(* CODESYS project sensata_vision.library
   Company: Sensata Technologies
   Version: 0.0.2
   DocFormat: reStructuredText
   Placeholder: Sensata_Vision
   Title: Sensata_Vision

Project tree, tasks and I/O mapping:
  libraries: Sensata_Common, * (Sensata Technologies); Sensata_IO, * (Sensata Technologies); Tc2_Standard, * (Beckhoff Automation GmbH); Tc2_System, * (Beckhoff Automation GmbH); Tc2_Utilities, * (Beckhoff Automation GmbH); Tc3_Module, * (Beckhoff Automation GmbH)
  Abstract/
    function block FB_BarcodeReader [ST]
    function block FB_Camera [ST]: M_SaveImage, P_bSaveImageBusy, M_ClearResults, M_ReadResult, P_bReadBusy, P_bResultsAvailable, M_Trigger, P_bTriggerBusy
  Concrete/
    Cognex/
      D900/
        data type E_CognexD900_Error
        function block FB_CognexD900 [ST]: P_strDescription, P_strMake, P_strModel, P_strVersion, M_Disable, M_Enable, M_GetEnableStatus, P_bEnableBusy, P_bEnabled, M_SaveImage, P_bSaveImageBusy, M_GetCurrentProgram, M_GetProgramState, M_LoadProgram, M_PauseProgram, M_StartProgram, M_StopProgram, P_bProgramControlBusy, P_enumProgramState, P_strCurrentProgram, M_ClearResults, M_ReadResult, P_bReadBusy, P_bResultsAvailable, M_Reset, P_bResetBusy, M_Trigger, P_bTriggerBusy
        data type ST_CognexD900_IO_Inputs
        data type ST_CognexD900_IO_Outputs
    Keyence/
      IX Series/
        function block FB_KeyenceIX_DLEC1A [ST]: M_Reset, P_bResetBusy, M_Trigger, P_bTriggerBusy, A_CommandRecovery, A_ControlsMapping, A_ValueMapping
        data type ST_KeyenceIXValue
      SR Series/
        Old/
          function block FB_KeyenceBarcodeReader [ST]: M_Disable, M_Enable, M_GetCurrentProgram, M_GetEnableStatus, M_GetProgramState, M_LoadProgram, M_PauseProgram, M_ReadResults, M_Reset, M_StartProgram, M_StopProgram, M_Trigger, P_bEnableBusy, P_bEnabled, P_bProgramControlBusy, P_bReadBusy, P_bResetBusy, P_bResultsAvailable, P_bTriggerBusy, P_enumProgramState, P_strCurrentProgram, P_strDescription, P_strMake, P_strModel, P_strVersion
          data type KeyenceSR700_Inputs
          data type KeyenceSR700_Outputs
        function block FB_KeyenceNL20_EIP [ST]: A_SR, M_ClearResults, M_ReadResult, M_Reset, M_Trigger, P_bReadBusy, P_bResetBusy, P_bResultsAvailable, P_bTriggerBusy
        function block FB_KeyenceSR [ST]: M_ClearResults, M_ReadResult, P_bReadBusy, P_bResultsAvailable, M_Reset, P_bResetBusy, M_Trigger, P_bTriggerBusy, A_ClearOutputs, A_CommandRecovery
        function block FB_KeyenceSR750_EIP [ST]: A_SR, M_ClearResults, M_ReadResult, M_Reset, M_Trigger, P_bReadBusy, P_bResetBusy, P_bResultsAvailable, P_bTriggerBusy
        function block FB_KeyenceSRX1H3H_EIP [ST]: A_SR, M_ClearResults, M_ReadResult, M_Reset, M_Trigger, P_bReadBusy, P_bResetBusy, P_bResultsAvailable, P_bTriggerBusy
  Interfaces/
    interface I_ImageSaving: M_SaveImage, P_bSaveImageBusy
    interface I_Readable: M_ClearResults, M_ReadResult, P_bReadBusy, P_bResultsAvailable
    interface I_Triggerable: M_Trigger, P_bTriggerBusy
  Project Information/
    function F_GetCompany [ST]
    function F_GetTitle [ST]
    function F_GetVersion [ST]
  Version/
    global variables Global_Version
*)

// Concrete/Cognex/D900/E_CognexD900_Error
{attribute 'qualified_only'}
{attribute 'strict'}
TYPE E_CognexD900_Error :
(
	NoError := 0,
	
	LoadProgramFail := 100,
	LoadRecipeFail := 101,
	
	TriggerTimeout := 200,
	
	ImageNameOrLocationTooLong := 300
) UDINT;
END_TYPE

// Concrete/Cognex/D900/ST_CognexD900_IO_Inputs
TYPE ST_CognexD900_IO_Inputs :
STRUCT
	bOnline : BOOL; (* Standard input from camera. TRUE when the camera is online. *)
	bReady : BOOL; (* Standard input from camera. TRUE when the camera is ready. *)
	bPaused : BOOL; (* Standard input from camera. TRUE when the camera is paused. *)
	bHasError : BOOL; (* Standard input from camera. TRUE when the camera has an error. *)
	intErrorCode : INT; (* Standard input from camera. Current error code. *)
	
	bTriggerReady : BOOL; (* Standard input from camera. TRUE when the trigger is ready. *)
	bTriggerAck : BOOL; (* Standard input from camera. Goes TRUE to acknowledge a trigger. *)
	bAcquisitionError : BOOL; (* Standard input from camera. Goes TRUE if acquisition failed. *)
	bExposureComplete : BOOL; (* Standard input from camera. Goes TRUE if exposure finished. *)
	
	bResultsValid : BOOL; (* Standard input from camera. Goes TRUE once inspection results are available. *)
	
	bCommandFailed : BOOL; (* Standard input from camera. TRUE if a command has failed. *)
	bCommandCompleted : BOOL; (* Standard input from camera. TRUE if a command has completed. *)
	
	bSetUserDataAck :  BOOL; (* Standard input from camera. Goes TRUE to acknowledge setting of user data buffer. *)

	bReadUserDataAck : BOOL; (* Should be assigned to an external trigger if image saving is used. *)
	bSaveImageAck : BOOL; (* Should be assigned to an external trigger if image saving is used. *)
END_STRUCT
END_TYPE

// Concrete/Cognex/D900/ST_CognexD900_IO_Outputs
TYPE ST_CognexD900_IO_Outputs :
STRUCT
	bTriggerEnable : BOOL; (* Standard output to camera. Set TRUE to enable trigger, FALSE to disable. *)
	bTrigger : BOOL; (* Standard output to camera. Rising edge to trigger camera. *)
	
	bResultAck : BOOL; (* Standard output to camera. Rising edge to acknowledge inspection result. *)
	
	bSetPaused : BOOL; (* Standard output to camera. Set TRUE to pause, FALSE to unpause. *)
	
	bClearError : BOOL; (* Standard output to camera. Rising edge to clear error. *)
	
	uintCommand : UINT; (* Standard output to camera. Set to a valid command ID before executing command. *)
	bExecuteCommand : BOOL; (* Standard output to camera. Set high to execute command. *)
	
	bSetUserData: BOOL; (* Standard output to camera. Set high to set user data buffer. *)
	
	bReadUserData : BOOL; (* Should be assigned to an external trigger if image saving is used. *)
	bSaveImage : BOOL; (* Should be set to an external trigger if image saving is enabled. *)
END_STRUCT
END_TYPE

// Concrete/Keyence/IX Series/ST_KeyenceIXValue
TYPE ST_KeyenceIXValue :
STRUCT
	bInvalid: BOOL;
	bUnderRange: BOOL;
	bOverRange: BOOL;
	dintValue: DINT;
END_STRUCT
END_TYPE

// Concrete/Keyence/SR Series/Old/KeyenceSR700_Inputs
TYPE KeyenceSR700_Inputs :
STRUCT
	Error								:BOOL;
	ResultDataAvailable					:BOOL;
	ResultDataStrobe					:BOOL;

	NoName0_arrBIT						:ARRAY[0..2] OF BOOL;
	NoName1_arrBIT						:ARRAY[0..2] OF BOOL;
	NoName2_arrBIT						:ARRAY[0..2] OF BOOL;
	NoName3_arrBIT						:ARRAY[0..2] OF BOOL;
	NoName4_arrBIT						:ARRAY[0..1] OF BOOL;
	NoName5_arrBIT						:BOOL;
	NoName6_arrBIT						:ARRAY[0..18] OF BOOL;

	NoName7_arrBYTE						:ARRAY[0..1] OF BYTE;
	NoName8_arrBYTE						:ARRAY[0..5] OF BYTE;
	NoName9_arrBYTE						:ARRAY[0..1] OF BYTE;
	NoName10_arrBYTE					:ARRAY[0..1] OF BYTE;


	BufferOverflowError					:BOOL;
	GeneralError						:BOOL;
	Busy								:BOOL;
	TRGBusy								:BOOL;
	LOCKBusy							:BOOL;
	ModeBusy							:BOOL;
	ErrorBusy							:BOOL;

	ReadComplete						:BOOL;
	PresetComplete						:BOOL;
	RegisterPresetDataComplete			:BOOL;
	TuneComplete						:BOOL;
	EXTRequestComplete					:BOOL;

	ReadFailure							:BOOL;
	PresetFailure						:BOOL;
	RegisterPresetDataFailure			:BOOL;
	TuneFailure							:BOOL;
	EXTRequestFailure					:BOOL;

	IN1Status							:BOOL;	
	IN2Status							:BOOL;	
	
	OUT1Status							:BOOL;	
	OUT2Status							:BOOL;	
	OUT3Status							:BOOL;	
		
	Unstable							:BOOL;
	MatchingLevel_Unstable				:BOOL;
	ISO_IEC15415_Unstable				:BOOL;
	AIM_DPM_Unstable					:BOOL;
	SAE_AS9132_Unstable					:BOOL;
	
	MatchingLevel						:UINT;
	ISO_IEC15415_Grade					:UINT;
	AIM_DPM_Grade						:UINT;

	ReadResultCode						:UINT;
	PresetResultCode					:UINT;
	RegisterPresetDataResultCode		:UINT;
	TuneResultCode						:UINT;
	EXTResquestResultCode				:UINT;
	GeneralErrorCode					:UINT;
	
	ResultData_ReadyCount				:UINT;
	ResultData_UpdateCount				:UINT;
	ResultData_Size						:UINT;
	ResultData							:ARRAY[0..128] OF BYTE;
	

END_STRUCT
END_TYPE

// Concrete/Keyence/SR Series/Old/KeyenceSR700_Outputs
TYPE KeyenceSR700_Outputs :
STRUCT

	ResultDataLatch						:BOOL;
	ClearError							:BOOL;

	ReadRequest							:BOOL;
	PresetRequest						:BOOL;
	RegisterPresetDataRequest			:BOOL;
	TuneRequest							:BOOL;

	ClearReadComplete					:BOOL;
	ClearPresetComplete					:BOOL;
	ClearRegisterPresetData				:BOOL;
	ClearTuneComplete					:BOOL;
	ClearEXTRequestComplete				:BOOL;

	BankNumber							:UINT;
	UserDataSize						:UINT;

	UserData							:ARRAY[0..64] OF BYTE;
	
	Noname0_BIT							:BOOL;
	Noname1_arrBIT						:ARRAY[0..4] OF BOOL;
	Noname2_arrBIT						:ARRAY[0..3] OF BOOL;
	Noname3_arrBIT						:ARRAY[0..2] OF BOOL;
	Noname4_BYTE						:BYTE;
	Noname5_arrBYTE						:ARRAY[0..3] OF BOOL;

END_STRUCT
END_TYPE

// Version/Global_Version
{attribute 'TcGenerated'}
{attribute 'no-analysis'}
{attribute 'linkalways'}
// This function has been automatically generated from the project information.
VAR_GLOBAL CONSTANT
	{attribute 'const_non_replaced'}
	stLibVersion_Sensata_Vision : ST_LibVersion := (iMajor := 0, iMinor := 0, iBuild := 2, iRevision := 0, nFlags := 0, sVersion := '0.0.2');
END_VAR

// Abstract/FB_BarcodeReader
FUNCTION_BLOCK ABSTRACT FB_BarcodeReader EXTENDS FB_Camera
VAR_INPUT
END_VAR
VAR_OUTPUT
END_VAR
VAR
END_VAR

END_FUNCTION_BLOCK

// Abstract/FB_Camera
(*
===============================================================================
Camera
===============================================================================
:Contact: Kevin Sanita <ksanita@sensata.com>
:Last Edited: December 2021

:Description: Represents a camera device.

:Notes:
* Standard use is to 
	1) Connect with I_Connectable
	2) Enable with I_Enableable
	3) Load program with I_Programmable
	4) Start program with I_Controllable
	5) While program is running, trigger with I_Triggerable
	6) Read inspect result with I_SimpleInspection

:Change Log:
- **December 20, 2021** Initial version
*)
FUNCTION_BLOCK ABSTRACT FB_Camera EXTENDS FB_Device
	IMPLEMENTS
		I_Triggerable, (* Most cameras will require triggering. *)
		I_Readable, (* Most cameras will require reading result data. *)
		I_ImageSaving (* Implements image saving functionality. *)
VAR_INPUT
END_VAR
VAR_OUTPUT
END_VAR
VAR
END_VAR

(* Saves an image with a specified name and save location. *)
METHOD M_SaveImage : BOOL
VAR_INPUT
	(* What to name the image file. *)
	strFilename	: Tc2_System.T_MaxString;
	(* Where to save the file, if applicable. *)
	strLocation	: Tc2_System.T_MaxString := '';
END_VAR
M_SaveImage := TRUE;
THIS^.M_LogWarning('M_SaveImage is not implemented!');
END_METHOD

PROPERTY P_bSaveImageBusy : BOOL
GET
P_bSaveImageBusy := FALSE;
END_GET
END_PROPERTY

(* Clears all results currently available on the camera. *)
METHOD M_ClearResults : BOOL
M_ClearResults := TRUE;
THIS^.M_LogWarning('Clear results not implemented!');
END_METHOD

(* Reads one result from the camera. *)
METHOD M_ReadResult : BOOL
M_ReadResult := TRUE;
THIS^.M_LogWarning('Read result not implemented!');
END_METHOD

(* True while this interface is busy. *)
PROPERTY P_bReadBusy : BOOL
GET
P_bReadBusy := FALSE;
END_GET
END_PROPERTY

(* True if there are results available. *)
PROPERTY P_bResultsAvailable : BOOL
GET
P_bResultsAvailable := FALSE;
END_GET
END_PROPERTY

(* Triggers the camera. *)
METHOD M_Trigger : BOOL
M_Trigger := TRUE;
THIS^.M_LogWarning('M_Trigger not implemented!');
END_METHOD

(* True while the camera is busy processing an image. *)
PROPERTY P_bTriggerBusy : BOOL
GET
P_bTriggerBusy := FALSE;
END_GET
END_PROPERTY

END_FUNCTION_BLOCK

// Interfaces/I_Triggerable
(*
===============================================================================
Triggerable
===============================================================================

:Description: Interface for modules that need to be triggered.

:Notes:
* Use ``M_Trigger`` to trigger the module.
* ``P_bTriggerBusy`` stays high while module is triggering. 
*)
INTERFACE I_Triggerable

(*
Triggers the function block.
*)
METHOD M_Trigger : BOOL
VAR_INPUT
END_VAR
END_METHOD

(*
Stays high while the function block is performing the tasks that were triggered.
*)
PROPERTY P_bTriggerBusy : BOOL
GET
END_GET
END_PROPERTY

END_INTERFACE

// Interfaces/I_Readable
(*
===============================================================================
Readable
===============================================================================

:Description: Interface for reading results data from inspection cameras.

:Notes:
* Use ``M_ReadResult`` to read result data from the camera.
* Use ``M_ClearResults`` to clear all results data.
* ``P_bReadBusy`` stays high while camera is being read. 
* ``P_bResultsAvailable`` is true if there is data available to read.
*)
INTERFACE I_Readable

(* Clears all results currently available on the camera. *)
METHOD M_ClearResults : BOOL
VAR_INPUT
END_VAR
END_METHOD

(* Reads one result from the camera. *)
METHOD M_ReadResult : BOOL
VAR_INPUT
END_VAR
END_METHOD

(* True while this interface is busy. *)
PROPERTY P_bReadBusy : BOOL
GET
END_GET
END_PROPERTY

(* True if there are results available. *)
PROPERTY P_bResultsAvailable : BOOL
GET
END_GET
END_PROPERTY

END_INTERFACE

// Interfaces/I_ImageSaving
INTERFACE I_ImageSaving

(* Saves an image with a specified name and save location. *)
METHOD M_SaveImage : BOOL
VAR_INPUT
	strFilename : T_MaxString; (* What to name the image file. *)
	strLocation : T_MaxString := ''; (* Where to save the file, if applicable. *)
END_VAR
END_METHOD

PROPERTY P_bSaveImageBusy : BOOL
GET
END_GET
END_PROPERTY

END_INTERFACE

// Concrete/Cognex/D900/FB_CognexD900
(*
===============================================================================
Function Block Name
===============================================================================
:Contact: Kevin Sanita <ksanita@sensata.com>
:Last Edited: January 2022

:Description: Cognex D900 implementation of FB_Camera

:Change Log:
- **January 4, 2021** Initial version
*)
FUNCTION_BLOCK FB_CognexD900 EXTENDS FB_Camera
	IMPLEMENTS 
		I_DeviceInfo, (* Required for all devices. *)
		I_Enableable, (* Cognex cameras have a trigger enable that must be set. *)
		I_Triggerable, (* The camera must be triggered to perform an inspection. *)
		I_Readable, (* Read results from the camera. *)
		I_Resettable, (* Need to be able to clear errors on the camera itself. *)
		I_Programmable, (* Must be able to load programs. *)
		I_ImageSaving (* Can use external triggers to save images. *)
VAR_INPUT
	stInputs : ST_CognexD900_IO_Inputs; (* Fieldbus inputs. *)
	arrUserData : REFERENCE TO ARRAY[0..487] OF BYTE; (* Standard output to camera. Contains user data for commands. *)
	
	(* Set to TRUE if image saving is enabled. Requires an event trigger to be
	set up in In-Sight Vision Suite. *)
	bImageSavingEnabled : BOOL; 
	uintImageFilenameOffset : UINT; (* User data location allocated to image filename. *)
	uintImageFilenameLength : UINT; (* User data length allocated to image filename. Set to zero to disable. *)
	uintImageLocationOffset : UINT; (* User data location allocated to image location. *)
	uintImageLocationLength : UINT; (* User data length allocated to image location. Set to zero to disable. *)
	
	// Program to load in format of job:recipe
	in_strProgram: T_MaxString;
END_VAR
VAR_OUTPUT
	stOutputs : ST_CognexD900_IO_Outputs; (* Fieldbus outputs. *)
END_VAR
VAR
	// Main
	fbErrorOccurred: R_TRIG; (* Rising edge trigger for errors. *)	

	// Control
	bControlBusy: BOOL; (* TRUE while pausing or unpausing camera program. *)
	
	// Trigger
	bTriggerBusy: BOOL; (* TRUE when the trigger is busy. *)
	
	// Read
	bReadBusy : BOOL; (* True while read is busy. *)
	
	// Reset
	bResetBusy: BOOL; (* TRUE when the camera is busy clearing error. *)
	
	// Load Program
	strRequestedProgram: STRING(255); (* The program request string containing job name or job and recipe separated by a colon. *)
	bProgramLoading: BOOL; (* TRUE while a job is loading. *)
	strRequestedJob: STRING(255); (* Requested job name. *)
	strRequestedRecipe: T_MaxString; (* Requested recipe name. *)
	intProgramLoadStep: INT; (* Current program loading step. *)
	intProgramRequestSplit: INT; (* Location of colon in program request string. *)
	strCurrentJob: T_MaxString; (* Currently loaded job *)
	strCurrentRecipe: T_MaxString; (* Currently loaded recipe. *)
	strCurrentProgram: T_MaxString; (* Currently loaded program. *)
	
	// Enable
	bEnableBusy: BOOL; (* TRUE while enable is busy. *)
	
	// Image saving
	bSaveImageBusy: BOOL; (* TRUE while image saving is busy. *)
	bUserDataSet: BOOL; (* TRUE if user data was set. *)
END_VAR

// Check camera for error.
fbErrorOccurred(CLK:=stInputs.bHasError);
IF fbErrorOccurred.Q THEN
	THIS^.M_SetError(INT_TO_UDINT(stInputs.intErrorCode), 'Camera error! Check camera documentation for error code details.');
END_IF

PROPERTY P_strDescription : Sensata_Common.T_MaxString
GET
P_strDescription := 'Cognex D900 Camera';
END_GET
END_PROPERTY

PROPERTY P_strMake : Sensata_Common.T_MaxString
GET
P_strMake := 'Cognex';
END_GET
END_PROPERTY

PROPERTY P_strModel : Sensata_Common.T_MaxString
GET
P_strModel := 'D900';
END_GET
END_PROPERTY

PROPERTY P_strVersion : Sensata_Common.T_MaxString
GET
END_GET
END_PROPERTY

(* Sets trigger enable low *)
METHOD M_Disable : BOOL
M_Disable := FALSE;
IF stOutputs.bTriggerEnable THEN
	bEnableBusy := TRUE;
	stOutputs.bTriggerEnable := FALSE;
	THIS^.M_LogMessage('Disabling trigger');
ELSIF NOT stInputs.bTriggerReady THEN
	IF bEnableBusy THEN
		bEnableBusy := FALSE;
		THIS^.M_LogMessage('Camera trigger disabled.');
	END_IF
	M_Disable := TRUE;
END_IF;
END_METHOD

(* Sets trigger enable high *)
METHOD M_Enable : BOOL
M_Enable := FALSE;
IF NOT stOutputs.bTriggerEnable THEN
	bEnableBusy := TRUE;
	stOutputs.bTriggerEnable := TRUE;
	THIS^.M_LogMessage('Enabling trigger');
ELSIF stInputs.bTriggerReady THEN
	IF bEnableBusy THEN
		bEnableBusy := FALSE;
		THIS^.M_LogMessage('Camera trigger enabled.');
	END_IF
	M_Enable := TRUE;
END_IF;
END_METHOD

(* Get the current enable status of the device. *)
METHOD M_GetEnableStatus : BOOL
VAR_OUTPUT
	bEnabled	: BOOL;
END_VAR
bEnabled := THIS^.P_bEnabled;
M_GetEnableStatus := TRUE;
END_METHOD

(* TRUE while the device is busy enabling or disabling. *)
PROPERTY P_bEnableBusy : BOOL
GET
P_bEnablebusy := bEnableBusy;
END_GET
END_PROPERTY

PROPERTY P_bEnabled : BOOL
GET
IF stInputs.bTriggerReady THEN
	P_bEnabled := TRUE;
ELSE
	P_bEnabled := FALSE;
END_IF
END_GET
END_PROPERTY

(* Saves an image with a specified name and save location. *)
METHOD M_SaveImage : BOOL
VAR_INPUT
	(* What to name the image file. *)
	strFilename	: Tc2_System.T_MaxString;
	(* Where to save the file, if applicable. *)
	strLocation	: Tc2_System.T_MaxString := '';
END_VAR

VAR
	bAbleToSave: BOOL;
	bFilenameValid: BOOL;
	bLocationValid: BOOL;
END_VAR
M_SaveImage := FALSE;

// Check that rest of camera isn't in a busy or error state
bAbleToSave := NOT THIS^.P_bError 
		AND NOT THIS^.P_bTriggerBusy
		AND NOT THIS^.P_bProgramControlBusy
		AND THIS^.P_enumProgramState = E_ProgramState.Running
		AND bImageSavingEnabled
		AND NOT bSaveImageBusy;

// If able to start saving, then try to start saving
IF bAbleToSave THEN
	
	// Check that the filename and location are not too long
	bFilenameValid := LEN(strFilename) < UINT_TO_INT(uintImageFilenameLength) OR uintImageFilenameLength = 0;
	bLocationValid := LEN(strLocation) < UINT_TO_INT(uintImageLocationLength) OR uintImageLocationLength = 0;
	
	IF bFilenameValid AND bLocationValid THEN
		// Send save image command
		bUserDataSet := FALSE;
		stOutputs.bSaveImage := FALSE;
		stOutputs.bSetUserData := FALSE;
		stOutputs.bReadUserData := FALSE;
		
		// Make sure the acknowledges are reset before starting trigger sequence
		IF NOT stInputs.bSaveImageAck AND NOT stInputs.bSetUserDataAck AND NOT stInputs.bReadUserDataAck THEN
			THIS^.M_LogMessage('Starting image save sequence.');
			bSaveImageBusy := TRUE;
		END_IF
	ELSE
		THIS^.M_SetError(
			E_CognexD900_Error.ImageNameOrLocationTooLong,
			'Filename or location for image saving is longer than allocated buffer space!');
	END_IF
	
// Wait for save image command to finish
ELSIF bSaveImageBusy THEN
	IF NOT bUserDataSet THEN
		IF NOT stOutputs.bSetUserData THEN
			// Save filename to user data buffer
			IF uintImageFilenameLength > 0 THEN
				MEMSET(ADR(arrUserData)+uintImageFilenameOffset, 0, uintImageFilenameLength);
				MEMCPY(ADR(arrUserData)+uintImageFilenameOffset, ADR(strFilename), INT_TO_UDINT(LEN(strFilename)));
			END_IF
			
			// Save location to user data sbuffer
			IF uintImageLocationLength > 0 THEN
				MEMSET(ADR(arrUserData)+uintImageLocationOffset, 0, uintImageLocationLength);
				MEMCPY(ADR(arrUserData)+uintImageLocationOffset, ADR(strLocation), INT_TO_UDINT(LEN(strLocation)));
			END_IF
		END_IF
		
		// Wait for user data to set.
		stOutputs.bSetUserData := TRUE;
		stOutputs.bReadUserData := TRUE;
		IF stInputs.bSetUserDataAck AND stInputs.bReadUserDataAck THEN
			THIS^.M_LogMessage('Set user data.');
			stOutputs.bReadUserData := FALSE;
			stOutputs.bSetUserData := FALSE;
			bUserDataSet := TRUE;
		END_IF
	ELSE
		// Wait for image to save
		stOutputs.bSaveImage := TRUE;
		IF stInputs.bSaveImageAck THEN
			THIS^.M_LogMessage('Image saved.');
			stOutputs.bSaveImage := FALSE;
			bSaveImageBusy := FALSE;
			M_SaveImage := TRUE;
		END_IF
	END_IF
END_IF
END_METHOD

PROPERTY P_bSaveImageBusy : BOOL
GET
P_bSaveImageBusy := bSaveImageBusy;
END_GET
END_PROPERTY

(* Gets the program currently loaded on the device. *)
METHOD M_GetCurrentProgram : BOOL
VAR_OUTPUT
	strCurrentProgram	: Sensata_Common.T_MaxString;
END_VAR
strCurrentProgram := THIS^.P_strCurrentProgram;
M_GetCurrentProgram := TRUE;
END_METHOD

(* Gets the current control state. *)
METHOD M_GetProgramState : BOOL
VAR_OUTPUT
	enumProgramState	: Sensata_Common.E_ProgramState;
END_VAR
enumProgramState := THIS^.P_enumProgramState;
M_GetProgramState := TRUE;
END_METHOD

 (*
Loads a new program on the module.
*)
METHOD M_LoadProgram : BOOL
M_LoadProgram := FALSE;

CASE intProgramLoadStep OF
	0: // Parse job and recipe
		bProgramLoading := TRUE;
		strRequestedProgram := in_strProgram;
		intProgramRequestSplit := FIND(strRequestedProgram, ':');
		IF intProgramRequestSplit > 0 THEN
			strRequestedJob := LEFT(strRequestedProgram, intProgramRequestSplit-1);
			strRequestedRecipe := RIGHT(strRequestedProgram, LEN(strRequestedProgram)-intProgramRequestSplit);
		ELSE
			strRequestedJob := strRequestedProgram;
			strRequestedRecipe := '';
		END_IF
		
		strCurrentProgram := '';
		
		intProgramLoadStep := intProgramLoadStep + 10;

	10: // Pause the camera
		IF THIS^.M_PauseProgram() THEN
			intProgramLoadStep := intProgramLoadStep + 10;
		END_IF
		
	20: // Send the load job by name command
		IF strCurrentJob <> strRequestedJob THEN
			// Set command to load program by name
			stOutputs.uintCommand := 16#4000; 

			// Copy program name to user data
			MEMSET(ADR(arrUserData), 0, SIZEOF(arrUserData));
			MEMCPY(ADR(arrUserData), ADR(strRequestedJob), INT_TO_UDINT(LEN(strRequestedJob)));
			
			// Set execute command bit
			stOutputs.bExecuteCommand := TRUE;
			
			THIS^.M_LogMessage('Loading job.');
			
			strCurrentJob := '';
			
			// Go to next step
			intProgramLoadStep := intProgramLoadStep + 10;
		ELSE
			intProgramLoadStep := intProgramLoadStep + 20;
		END_IF
		
	30: // Wait for command to complete
		IF stInputs.bCommandCompleted THEN
			stOutputs.bExecuteCommand := FALSE;
			IF stInputs.bCommandFailed THEN
				THIS^.M_SetError(E_CognexD900_Error.LoadProgramFail, 'Failed to load job!.');
				bProgramLoading := FALSE;
				intProgramLoadStep := 0;
			END_IF
		ELSIF NOT stOutputs.bExecuteCommand THEN
			THIS^.M_LogMessage('Finished loading job.');
			strCurrentJob := strRequestedJob;
			intProgramLoadStep := intProgramLoadStep + 10;
		END_IF
		
	40: // Send the load recipe by name command

		IF LEN(strRequestedRecipe) > 0 AND strRequestedRecipe <> strCurrentRecipe THEN
			// Set command to load recipe by name
			stOutputs.uintCommand := 16#4001; 

			// Copy program name to user data
			MEMSET(ADR(arrUserData), 0, SIZEOF(arrUserData));
			MEMCPY(ADR(arrUserData), ADR(strRequestedRecipe), INT_TO_UDINT(LEN(strRequestedRecipe)));
			
			// Set execute command bit
			stOutputs.bExecuteCommand := TRUE;
			
			THIS^.M_LogMessage('Loading recipe.');
			
			strCurrentRecipe := '';
			
			// Go to next step
			intProgramLoadStep := intProgramLoadStep + 10;
		ELSE
			intProgramLoadStep := intProgramLoadStep + 20;
		END_IF

		
	50: // Wait for command to complete
		IF stInputs.bCommandCompleted THEN
			stOutputs.bExecuteCommand := FALSE;
			IF stInputs.bCommandFailed THEN
				THIS^.M_SetError(E_CognexD900_Error.LoadRecipeFail, 'Failed to load recipe!.');
				bProgramLoading := FALSE;
				intProgramLoadStep := 0;
			END_IF
		ELSIF NOT stOutputs.bExecuteCommand THEN
			THIS^.M_LogMessage('Finished loading recipe.');
			strCurrentRecipe := strRequestedRecipe;
			intProgramLoadStep := intProgramLoadStep + 10;
		END_IF
	
	60: // Unpause the camera
		strCurrentProgram := strRequestedProgram;
		IF THIS^.M_StartProgram() THEN
			intProgramLoadStep := 0;
			bProgramLoading := FALSE;
			M_LoadProgram := TRUE;
		END_IF
END_CASE
END_METHOD

(*
Pauses the D900
*)
METHOD M_PauseProgram : BOOL
M_PauseProgram := FALSE;
IF NOT stInputs.bOnline THEN
	IF stOutputs.bSetPaused AND bControlBusy THEN
		THIS^.M_LogMessage('Camera paused.');
		bControlBusy := FALSE;
	END_IF
	M_PauseProgram := TRUE;
ELSE
	IF NOT stOutputs.bSetPaused THEN
		stOutputs.bSetPaused := TRUE;
		bControlBusy := TRUE;
		THIS^.M_LogMessage('Pausing camera.');
	END_IF
END_IF
END_METHOD

(*
Unpauses the D900
*)
METHOD M_StartProgram : BOOL
IF stInputs.bOnline AND NOT stOutputs.bSetPaused THEN
	IF bControlBusy THEN
		bControlBusy := FALSE;
		THIS^.M_LogMessage('Camera started.');
	END_IF
	M_StartProgram := TRUE;
ELSE
	IF stOutputs.bSetPaused THEN
		THIS^.M_LogMessage('Starting the camera.');
		stOutputs.bSetPaused := FALSE;
		bControlBusy := TRUE;
	END_IF
END_IF
END_METHOD

(*
Pauses the D900
*)
METHOD M_StopProgram : BOOL
M_StopProgram := THIS^.M_PauseProgram();
END_METHOD

(*
TRUE while a program is being loaded
*)
PROPERTY P_bProgramControlBusy : BOOL
GET
P_bProgramControlBusy := bProgramLoading OR bControlBusy;
END_GET
END_PROPERTY

(*
The current ``I_Controllable`` control state of the device
*)
PROPERTY P_enumProgramState : Sensata_Common.E_ProgramState
GET
IF stInputs.bPaused AND NOT stInputs.bOnline THEN
	P_enumProgramState := E_ProgramState.Paused;
ELSIF NOT stInputs.bOnline THEN
	P_enumProgramState := E_ProgramState.Stopped;
ELSE
	P_enumProgramState := E_ProgramState.Running;
END_IF
END_GET
END_PROPERTY

(*
The currently loaded program
*)
PROPERTY P_strCurrentProgram : Sensata_Common.T_MaxString
GET
P_strCurrentProgram := strCurrentProgram;
END_GET
END_PROPERTY

(* Clears all results currently available on the camera. *)
METHOD M_ClearResults : BOOL
// Clear out results
M_ClearResults := FALSE;
IF NOT bReadBusy AND NOT bTriggerBusy THEN
	// Acknowledge result if there are results
	IF stInputs.bResultsValid THEN
		THIS^.M_LogMessage('Clearing results.');
		stOutputs.bResultAck := TRUE;
		bReadBusy := TRUE;
	ELSE
		M_ClearResults := TRUE;
	END_IF
ELSIF stOutputs.bResultAck THEN
	// Wait for results to clear
	IF NOT stInputs.bResultsValid THEN
		THIS^.M_LogMessage('Results cleared.');
		stOutputs.bResultAck := FALSE;
		M_ClearResults := TRUE;
		bReadBusy := FALSE;
	END_IF
END_IF
END_METHOD

(* Reads one result from the camera. *)
METHOD M_ReadResult : BOOL

VAR
	bAbleToRead: BOOL;
END_VAR
M_ReadResult := FALSE;

bAbleToRead := NOT bTriggerBusy AND NOT bReadBusy AND stInputs.bResultsValid;

IF bAbleToRead THEN
	bReadBusy := TRUE;
	THIS^.M_LogMessage('Results received.');
	stOutputs.bResultAck := TRUE;
ELSIF stOutputs.bResultAck AND NOT stInputs.bResultsValid THEN
	THIS^.M_LogMessage('Results acknowledged.');
	bReadBusy := FALSE;
	stOutputs.bResultAck := FALSE;
	M_ReadResult := TRUE;
END_IF
END_METHOD

(* True while this interface is busy. *)
PROPERTY P_bReadBusy : BOOL
GET
P_bReadBusy := bReadBusy;
END_GET
END_PROPERTY

(* True if there are results available. *)
PROPERTY P_bResultsAvailable : BOOL
GET
P_bResultsAvailable := stInputs.bResultsValid;
END_GET
END_PROPERTY

(* Resets the module and clears any external errors. *)
METHOD M_Reset : BOOL
M_Reset := FALSE;
IF NOT stInputs.bHasError THEN
	IF bResetBusy THEN
		THIS^.M_LogMessage('Error cleared.');
		THIS^.M_ClearError();
		stOutputs.bClearError := FALSE;
		
		intProgramLoadStep := 0;
		bProgramLoading := FALSE;
		
		bResetBusy := FALSE;
		bTriggerBusy := FALSE;
		bControlBusy := FALSE;
		bReadBusy := FALSE;
		bSaveImageBusy := FALSE;
		
	END_IF
	M_Reset := TRUE;
ELSE 
	IF NOT bResetBusy THEN
		bResetBusy := TRUE;
		stOutputs.bClearError := TRUE;
		THIS^.M_LogMessage('Clearing error.');
	END_IF
END_IF
END_METHOD

(* Stays high while module is resetting. *)
PROPERTY P_bResetBusy : BOOL
GET
P_bResetBusy := bResetBusy;
END_GET
END_PROPERTY

(*
Triggers the function block.
*)
METHOD M_Trigger : BOOL
VAR
	bAbleToTrigger: BOOL;
END_VAR
M_Trigger := FALSE;

bAbleToTrigger := THIS^.P_enumProgramState = E_ProgramState.Running
	AND NOT bTriggerBusy AND NOT bReadBusy AND stInputs.bTriggerReady;

IF bAbleToTrigger THEN
	THIS^.M_LogMessage('Triggering.');
	stOutputs.bTrigger := FALSE;
	bTriggerBusy := TRUE;
ELSIF bTriggerBusy THEN
	stOutputs.bTrigger := TRUE;
	IF stInputs.bExposureComplete AND stInputs.bTriggerAck THEN
		THIS^.M_LogMessage('Trigger complete.');
		stOutputs.bTrigger := FALSE;
		bTriggerBusy := FALSE;
		M_Trigger := TRUE;
	ELSIF stInputs.bAcquisitionError AND stInputs.bTriggerAck THEN
		THIS^.M_LogMessage('Trigger error.');
		stOutputs.bTrigger := FALSE;
		bTriggerBusy := FALSE;
	END_IF
END_IF
END_METHOD

(*
Stays high while the function block is performing the tasks that were triggered.
*)
PROPERTY P_bTriggerBusy : BOOL
GET
P_bTriggerBusy := bTriggerBusy;
END_GET
END_PROPERTY

END_FUNCTION_BLOCK

// Concrete/Keyence/IX Series/FB_KeyenceIX_DLEC1A
FUNCTION_BLOCK FB_KeyenceIX_DLEC1A EXTENDS FB_Camera
	IMPLEMENTS I_Triggerable, I_Resettable, I_Resettable
VAR_INPUT
	// Set to TRUE if using the DLEC1A expansion channel and not main channel
	in_bExpansion: BOOL;
	// Program number to load when calling M_LoadProgram. Must be between 0 and 15.
	in_uintProgNumRequest: UINT(0..15);
END_VAR
VAR_IN_OUT
	// DLEC1A IO connection
	inout_stIO: ST_DLEC1A;
END_VAR
VAR_OUTPUT
	// Array of output values from the DLEC1A unit
	out_arrValues: ARRAY[1..8] OF ST_KeyenceIXValue;
	// Array of user output bits from the sensor
	out_arrOutputs: ARRAY[1..10] OF BOOL;
END_VAR
VAR
	// Index for iterations
	intIndex: INT;
	
	// Controls
	// Set to TRUE to trigger the height check
	bTriggerRequest: BOOL;
	// Gets set to TRUE when the trigger request is acknowledged
	bTriggerAck: BOOL;
	// Alternates between TRUE and FALSE as triggers are read
	bValueUpdate: BOOL;
	// Set to TRUE to load program number in_uintProgNumRequest
	bProgChangeRequest: BOOL;
	// Gets set to TRUE once program change is complete
	bProgChangeAck: BOOL;
	// Set to TRUE to set the offset
	bZeroOffsetRequest: BOOL;
	// Gets set to TRUE when zero/offset is complete
	bZeroOffsetAck: BOOL;
	// TRUE if there is an error
	bError: BOOL;
	// TRUE if there is a warning
	bWarning: BOOL;
	// Set TRUE to reset. No Ack, use bValueUpdate to capture completion.
	bResetRequest: BOOL;
	// Set TRUE to request an emission stop
	bEmissionStopRequest: BOOL;
	// Gets set to TRUE when emission stop is active
	bEmissionStopAck: BOOL;
	
	// Internal variables
	
	// TRUE while triggering
	bTriggering: BOOL;

	// TRUE while M_Trigger is running
	bTriggerBusy: BOOL;
	// Current M_Trigger step
	intTriggerStep: INT;
END_VAR

A_ValueMapping();
A_ControlsMapping();
A_CommandRecovery();

(* This should clear any errors on the device and bring it to a state where
	it is ready to be energized or otherwise activated. *)
METHOD M_Reset : BOOL
bTriggerRequest := FALSE;
bZeroOffsetRequest := FALSE;
bResetRequest := FALSE;
bProgChangeRequest := FALSE;
M_Reset := TRUE;
THIS^.M_LogMessage('Reset outputs');
END_METHOD

(* This property should be TRUE while any method in this interface is actively
	executing, or FALSE otherwise. *)
PROPERTY P_bResetBusy : BOOL
GET
P_bResetBusy := FALSE;
END_GET
END_PROPERTY

(*
Triggers the function block.
*)
METHOD M_Trigger : BOOL

VAR_INST
	_inst_bLastValue: BOOL;
END_VAR
VAR_INST // added by the converter: edge detectors and wires of the graphical bodies
    _w1, _w2, _w3, _w4, _w5, _w6, _w7, _w8, _w9, _w10 : BOOL;
    _rt1 : R_TRIG;
END_VAR
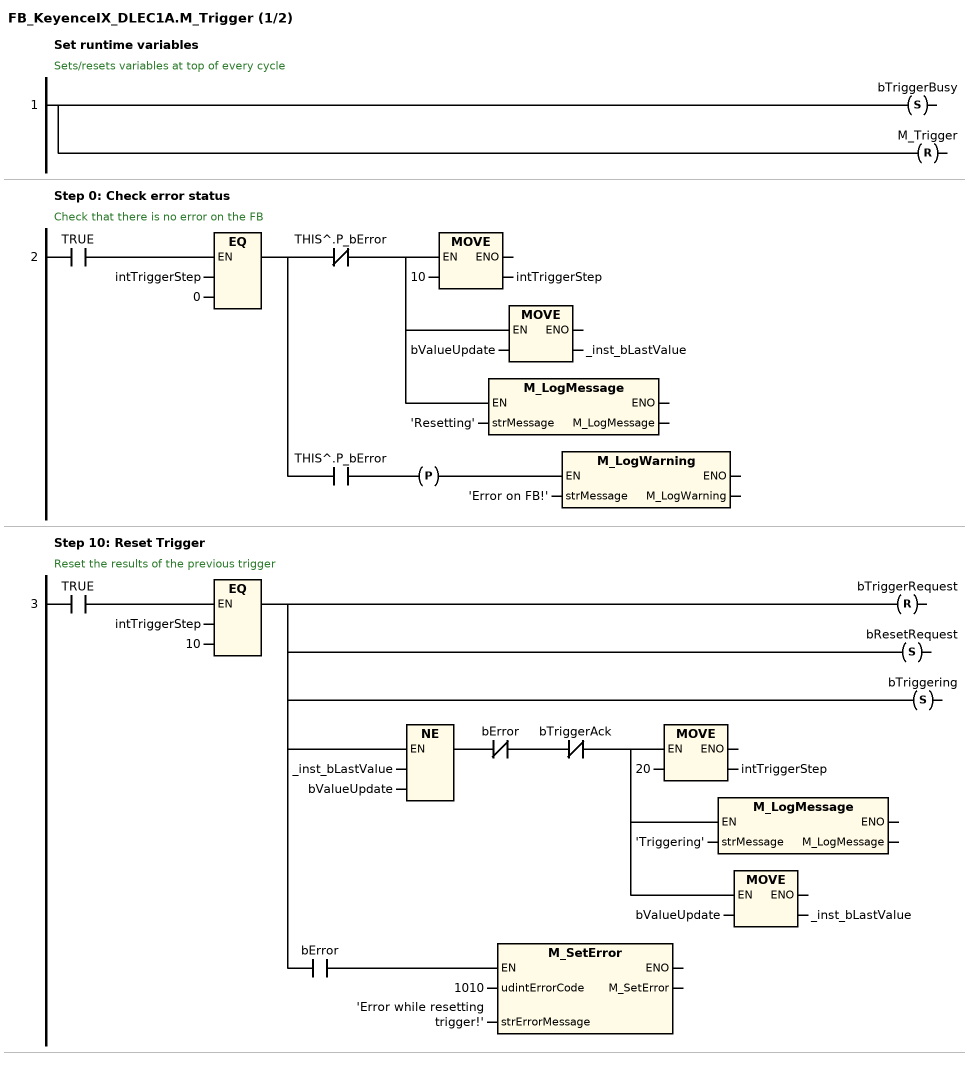
// NETWORK 1: Set runtime variables
// Sets/resets variables at top of every cycle
bTriggerBusy S= TRUE;
M_Trigger R= TRUE;

// NETWORK 2: Step 0: Check error status
// Check that there is no error on the FB
_w1 := intTriggerStep = 0;
_w2 := _w1 AND NOT THIS^.P_bError;
IF _w2 THEN intTriggerStep := 10; END_IF
IF _w2 THEN _inst_bLastValue := bValueUpdate; END_IF
IF _w2 THEN M_LogMessage(strMessage := 'Resetting'); END_IF
_rt1(CLK := _w1 AND THIS^.P_bError);
IF _rt1.Q THEN M_LogWarning(strMessage := 'Error on FB!'); END_IF

// NETWORK 3: Step 10: Reset Trigger
// Reset the results of the previous trigger
_w3 := intTriggerStep = 10;
bTriggerRequest R= _w3;
bResetRequest S= _w3;
bTriggering S= _w3;
_w4 := (_w3 AND _inst_bLastValue <> bValueUpdate) AND NOT bError AND NOT bTriggerAck;
IF _w4 THEN intTriggerStep := 20; END_IF
IF _w4 THEN M_LogMessage(strMessage := 'Triggering'); END_IF
IF _w4 THEN _inst_bLastValue := bValueUpdate; END_IF
IF _w3 AND bError THEN
    M_SetError(udintErrorCode := 1010, strErrorMessage := 'Error while resetting trigger!');
END_IF

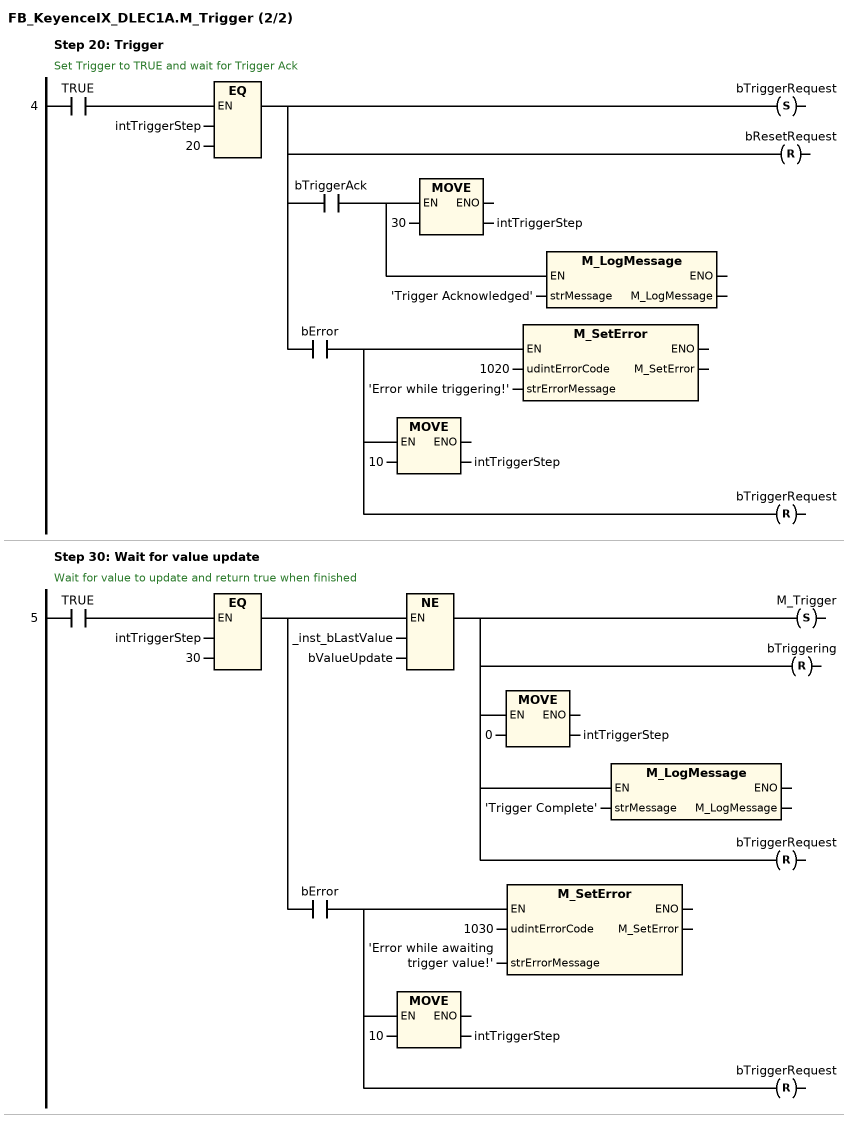
// NETWORK 4: Step 20: Trigger
// Set Trigger to TRUE and wait for Trigger Ack
_w5 := intTriggerStep = 20;
bTriggerRequest S= _w5;
bResetRequest R= _w5;
_w6 := _w5 AND bTriggerAck;
IF _w6 THEN intTriggerStep := 30; END_IF
IF _w6 THEN M_LogMessage(strMessage := 'Trigger Acknowledged'); END_IF
_w7 := _w5 AND bError;
IF _w7 THEN M_SetError(udintErrorCode := 1020, strErrorMessage := 'Error while triggering!'); END_IF
IF _w7 THEN intTriggerStep := 10; END_IF
bTriggerRequest R= _w7;

// NETWORK 5: Step 30: Wait for value update
// Wait for value to update and return true when finished
_w8 := intTriggerStep = 30;
_w9 := _w8 AND _inst_bLastValue <> bValueUpdate;
M_Trigger S= _w9;
bTriggering R= _w9;
IF _w9 THEN intTriggerStep := 0; END_IF
IF _w9 THEN M_LogMessage(strMessage := 'Trigger Complete'); END_IF
bTriggerRequest R= _w9;
_w10 := _w8 AND bError;
IF _w10 THEN M_SetError(udintErrorCode := 1030, strErrorMessage := 'Error while awaiting trigger value!'); END_IF
IF _w10 THEN intTriggerStep := 10; END_IF
bTriggerRequest R= _w10;
END_METHOD

(*
Stays high while the function block is performing the tasks that were triggered.
*)
PROPERTY P_bTriggerBusy : BOOL
GET
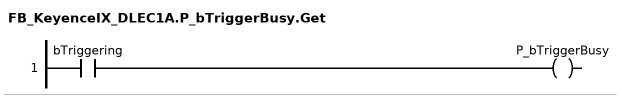
// NETWORK 1
P_bTriggerBusy := bTriggering;
END_GET
END_PROPERTY

ACTION A_CommandRecovery:
IF NOT bTriggerBusy AND intTriggerStep > 0 THEN
	intTriggerStep := 0;
	bTriggerRequest := FALSE;
	bTriggering := FALSE;
	THIS^.M_LogWarning('M_Trigger ended prematurely!');
END_IF
bTriggerBusy := FALSE;
END_ACTION

ACTION A_ControlsMapping:
IF in_bExpansion THEN
	bTriggerAck := BIT_TO_BOOL(inout_stIO.stIn.stResponse.bitExpTriggerAck);
	bValueUpdate := BIT_TO_BOOL(inout_stIO.stIn.stResponse.bitExpValueUpdateAck);
	bProgChangeAck := BIT_TO_BOOL(inout_stIO.stIn.stResponse.bitExpProgChgAck);
	bZeroOffsetAck := BIT_TO_BOOL(inout_stIO.stIn.stResponse.bitExpZeroOffsetAck);
	bEmissionStopAck := BIT_TO_BOOL(inout_stIO.stIn.stResponse.bitExpEmissionStopAck);
	bError := BIT_TO_BOOL(inout_stIO.stIn.stResponse.bitExpError);
	bWarning := BIT_TO_BOOL(inout_stIO.stIn.stResponse.bitExpWarning);

	out_arrOutputs[01] := BIT_TO_BOOL(inout_stIO.stIn.stResponse.bitExpOutput01);
	out_arrOutputs[02] := BIT_TO_BOOL(inout_stIO.stIn.stResponse.bitExpOutput02);
	out_arrOutputs[03] := BIT_TO_BOOL(inout_stIO.stIn.stResponse.bitExpOutput03);
	out_arrOutputs[04] := BIT_TO_BOOL(inout_stIO.stIn.stResponse.bitExpOutput04);
	out_arrOutputs[05] := BIT_TO_BOOL(inout_stIO.stIn.stResponse.bitExpOutput05);
	out_arrOutputs[06] := BIT_TO_BOOL(inout_stIO.stIn.stResponse.bitExpOutput06);
	out_arrOutputs[07] := BIT_TO_BOOL(inout_stIO.stIn.stResponse.bitExpOutput07);
	out_arrOutputs[08] := BIT_TO_BOOL(inout_stIO.stIn.stResponse.bitExpOutput08);
	out_arrOutputs[09] := BIT_TO_BOOL(inout_stIO.stIn.stResponse.bitExpOutput09);
	out_arrOutputs[10] := BIT_TO_BOOL(inout_stIO.stIn.stResponse.bitExpOutput10);

	inout_stIO.stOut.stRequest.bitExpTrigger := bTriggerRequest;
	inout_stIO.stOut.stRequest.bitExpProgChange := bProgChangeRequest;
	inout_stIO.stOut.stRequest.bitExpZeroOffset := bZeroOffsetRequest;
	inout_stIO.stOut.stRequest.bitExpReset := bResetRequest;
	inout_stIO.stOut.stRequest.bitExpEmissionStop := bEmissionStopRequest;
	inout_stIO.stOut.stRequest.bitExpProgNumBit0 := in_uintProgNumRequest.0;
	inout_stIO.stOut.stRequest.bitExpProgNumBit1 := in_uintProgNumRequest.1;
	inout_stIO.stOut.stRequest.bitExpProgNumBit2 := in_uintProgNumRequest.2;
	inout_stIO.stOut.stRequest.bitExpProgNumBit3 := in_uintProgNumRequest.3;
ELSE
	bTriggerAck := BIT_TO_BOOL(inout_stIO.stIn.stResponse.bitMainTriggerAck);
	bValueUpdate := BIT_TO_BOOL(inout_stIO.stIn.stResponse.bitMainValueUpdateAck);
	bProgChangeAck := BIT_TO_BOOL(inout_stIO.stIn.stResponse.bitMainProgChgAck);
	bZeroOffsetAck := BIT_TO_BOOL(inout_stIO.stIn.stResponse.bitMainZeroOffsetAck);
	bEmissionStopAck := BIT_TO_BOOL(inout_stIO.stIn.stResponse.bitMainEmissionStopAck);
	bError := BIT_TO_BOOL(inout_stIO.stIn.stResponse.bitMainError);
	bWarning := BIT_TO_BOOL(inout_stIO.stIn.stResponse.bitMainWarning);
	
	out_arrOutputs[01] := BIT_TO_BOOL(inout_stIO.stIn.stResponse.bitMainOutput01);
	out_arrOutputs[02] := BIT_TO_BOOL(inout_stIO.stIn.stResponse.bitMainOutput02);
	out_arrOutputs[03] := BIT_TO_BOOL(inout_stIO.stIn.stResponse.bitMainOutput03);
	out_arrOutputs[04] := BIT_TO_BOOL(inout_stIO.stIn.stResponse.bitMainOutput04);
	out_arrOutputs[05] := BIT_TO_BOOL(inout_stIO.stIn.stResponse.bitMainOutput05);
	out_arrOutputs[06] := BIT_TO_BOOL(inout_stIO.stIn.stResponse.bitMainOutput06);
	out_arrOutputs[07] := BIT_TO_BOOL(inout_stIO.stIn.stResponse.bitMainOutput07);
	out_arrOutputs[08] := BIT_TO_BOOL(inout_stIO.stIn.stResponse.bitMainOutput08);
	out_arrOutputs[09] := BIT_TO_BOOL(inout_stIO.stIn.stResponse.bitMainOutput09);
	out_arrOutputs[10] := BIT_TO_BOOL(inout_stIO.stIn.stResponse.bitMainOutput10);
	
	inout_stIO.stOut.stRequest.bitMainTrigger := bTriggerRequest;
	inout_stIO.stOut.stRequest.bitMainProgChange := bProgChangeRequest;
	inout_stIO.stOut.stRequest.bitMainZeroOffset := bZeroOffsetRequest;
	inout_stIO.stOut.stRequest.bitMainReset := bResetRequest;
	inout_stIO.stOut.stRequest.bitMainEmissionStop := bEmissionStopRequest;
	inout_stIO.stOut.stRequest.bitMainProgNumBit0 := in_uintProgNumRequest.0;
	inout_stIO.stOut.stRequest.bitMainProgNumBit1 := in_uintProgNumRequest.1;
	inout_stIO.stOut.stRequest.bitMainProgNumBit2 := in_uintProgNumRequest.2;
	inout_stIO.stOut.stRequest.bitMainProgNumBit3 := in_uintProgNumRequest.3;
END_IF
END_ACTION

ACTION A_ValueMapping:
FOR intIndex := 1 TO 8 DO
	out_arrValues[intIndex].dintValue := inout_stIO.stIn.arrCurrentValue[intIndex];
END_FOR

out_arrValues[1].bInvalid := BIT_TO_BOOL(inout_stIO.stIn.stResponse.bitValue1Invalid);
out_arrValues[1].bUnderRange := BIT_TO_BOOL(inout_stIO.stIn.stResponse.bitValue1UnderRange);
out_arrValues[1].bOverRange := BIT_TO_BOOL(inout_stIO.stIn.stResponse.bitValue1OverRange);

out_arrValues[2].bInvalid := BIT_TO_BOOL(inout_stIO.stIn.stResponse.bitValue2Invalid);
out_arrValues[2].bUnderRange := BIT_TO_BOOL(inout_stIO.stIn.stResponse.bitValue2UnderRange);
out_arrValues[2].bOverRange := BIT_TO_BOOL(inout_stIO.stIn.stResponse.bitValue2OverRange);

out_arrValues[3].bInvalid := BIT_TO_BOOL(inout_stIO.stIn.stResponse.bitValue3Invalid);
out_arrValues[3].bUnderRange := BIT_TO_BOOL(inout_stIO.stIn.stResponse.bitValue3UnderRange);
out_arrValues[3].bOverRange := BIT_TO_BOOL(inout_stIO.stIn.stResponse.bitValue3OverRange);

out_arrValues[4].bInvalid := BIT_TO_BOOL(inout_stIO.stIn.stResponse.bitValue4Invalid);
out_arrValues[4].bUnderRange := BIT_TO_BOOL(inout_stIO.stIn.stResponse.bitValue4UnderRange);
out_arrValues[4].bOverRange := BIT_TO_BOOL(inout_stIO.stIn.stResponse.bitValue4OverRange);

out_arrValues[5].bInvalid := BIT_TO_BOOL(inout_stIO.stIn.stResponse.bitValue5Invalid);
out_arrValues[5].bUnderRange := BIT_TO_BOOL(inout_stIO.stIn.stResponse.bitValue5UnderRange);
out_arrValues[5].bOverRange := BIT_TO_BOOL(inout_stIO.stIn.stResponse.bitValue5OverRange);

out_arrValues[6].bInvalid := BIT_TO_BOOL(inout_stIO.stIn.stResponse.bitValue6Invalid);
out_arrValues[6].bUnderRange := BIT_TO_BOOL(inout_stIO.stIn.stResponse.bitValue6UnderRange);
out_arrValues[6].bOverRange := BIT_TO_BOOL(inout_stIO.stIn.stResponse.bitValue6OverRange);

out_arrValues[7].bInvalid := BIT_TO_BOOL(inout_stIO.stIn.stResponse.bitValue7Invalid);
out_arrValues[7].bUnderRange := BIT_TO_BOOL(inout_stIO.stIn.stResponse.bitValue7UnderRange);
out_arrValues[7].bOverRange := BIT_TO_BOOL(inout_stIO.stIn.stResponse.bitValue7OverRange);

out_arrValues[8].bInvalid := BIT_TO_BOOL(inout_stIO.stIn.stResponse.bitValue8Invalid);
out_arrValues[8].bUnderRange := BIT_TO_BOOL(inout_stIO.stIn.stResponse.bitValue8UnderRange);
out_arrValues[8].bOverRange := BIT_TO_BOOL(inout_stIO.stIn.stResponse.bitValue8OverRange);
END_ACTION

END_FUNCTION_BLOCK

// Concrete/Keyence/SR Series/Old/FB_KeyenceBarcodeReader
{obsolete 'Use FB_KeyenceSR or a derivative of it!'}
FUNCTION_BLOCK FB_KeyenceBarcodeReader EXTENDS FB_BarcodeReader

	IMPLEMENTS 

		I_DeviceInfo, (* Required for all devices. *)
		I_Enableable, (* Cognex cameras have a trigger enable that must be set. *)
		I_Resettable, (* Need to be able to clear errors on the camera itself. *)
		I_Programmable (* Must be able to load programs. *)

VAR_INPUT

		// Triggr to barcode for Read from Staion step
		bTrigger: BOOL;

		// Reset the results Command FROM PLC
		bReset: BOOL;

		// Read complete signal from Barcode Reader
		in_bReadComplete: BOOL;

		// Result data available from Barcode reader
		in_bResultDataAvailable: BOOL;

		// Out 1 result from Barcode reader
		in_bOut1Results: BOOL;

		// Barcode Output 2 which is bad read
		in_bOut2Results: BOOL;

		// Fail to read status from Barcode
		in_bOut3Results: BOOL;
		
		
		in_uintReadDataSize: UINT;
		
	
		//String from Server data
		in_arrReadData: ARRAY[0..128] OF BYTE;	

END_VAR
VAR_OUTPUT

		// Trigger to barcode reader
		out_bReadRequest: BOOL;		

		// Out reset signals to Barcode reader
		out_ErrorClear:BOOL;
		out_ReadCompleteClear:BOOL;
		out_PresetCompleteClear:BOOL;
		out_EXTRequestCompleteClear:BOOL;

		// Clearring data available signal from PLC to Barcode
		out_RegisterPresetClearDataAvailable: BOOL;	

		//Preset Input Data bit 
//		out_PresetRequest: BOOL;
//		out_RegisterPresetDataRequest:BOOL;	
			
		// Barcode read results Good
		out_BarcodeReadGood: BOOL;
		
		// Barcode read Bad
		out_BarcodeReadBadORError: BOOL;
		
		// Read Data From Keyence
		out_strReadData: STRING(128);

			
END_VAR
VAR
		CameraTriggerTP: TP;
		TriggerCounter: CTU;
		PresetTimerReq: TON;
		PresetTrig: R_TRIG;	
		ReadCompleteTrig: R_TRIG;

		ResetCase: INT;
		TriggerCAse: INT;	
		Readcase: INT;	

		Test: BOOL;
		b_BusyTrigger: BOOL;
		bReadBusy: BOOL;
			CaeraTrigDelay: TON;

		bResetBusy: BOOL;
END_VAR

(* This method should return to the device to the state it was prior to being
	enabled. P_bEnabled should be immediately set to false unless the status of
	the device is explicitly known to still be enabled. After being disabled,
	the device should typically be unable to perform process steps. Once
	successfully disabled, this method should return TRUE. *)
METHOD M_Disable : BOOL
END_METHOD

(* This method should perform any tasks that must be performed after a device
	is energized, but prior to the device being used in a process, and then
	return TRUE and set P_bEnabled to TRUE once those tasks are completed. *)
METHOD M_Enable : BOOL
END_METHOD

(* This method should explicitly get the current program loaded on the device.
	If the current program is successfully gotten, this method should return
	TRUE and set P_strCurrentProgram and strCurrentProgram to the gotten
	program name. If this method fails, both should be set to empty strings. *)
METHOD M_GetCurrentProgram : BOOL
VAR_OUTPUT
	(* This should be set to the name of the currently loaded program if
		the method was successful, or a blank string otherwise. *)
	strCurrentProgram	: Sensata_Common.T_MaxString;
END_VAR
END_METHOD

(* This method should explicitly check the enable status of the device.
	Once the enable status is known, this method should return TRUE.
	If this method fails, P_bEnabled should be set to FALSE since the device
	is not absolutely known to still be enabled. *)
METHOD M_GetEnableStatus : BOOL
VAR_OUTPUT
	(* This should return TRUE if the device is explicitly known to be
		enabled, or FALSE otherwise. *)
	bEnabled	: BOOL;
END_VAR
END_METHOD

(* This method should explicitly check the program state of the device.
	Once the program state is known, this method should return TRUE and set
	P_enumProgramState and enumProgramState to the relevant E_ProgramState
	value, else it should set both to E_ProgramState.Unknown. *)
METHOD M_GetProgramState : BOOL
VAR_OUTPUT
	(* If the program state is successfully gotten, this should be set to
		the relevant E_ProgramState value. If this method fails, this should
		be set to E_ProgramState.Unknown. *)
	enumProgramState	: Sensata_Common.E_ProgramState;
END_VAR
END_METHOD

(* This method should load a new program onto the device, and then return TRUE
	once program loading is completed. Once this method begins the program loading
	process, P_strCurrentProgram should be cleared unless it is still explicitly
	known to be loaded. *)
METHOD M_LoadProgram : BOOL
END_METHOD

(* This program should move to the program state from whatever state it was in
	to the Paused state, and then return TRUE once successful. If the program
	state is Stopped, this method should return TRUE but keep the current state
	as Stopped, since Paused at the beginning at the program is equivalent to
	being Stopped. *)
METHOD M_PauseProgram : BOOL
END_METHOD

METHOD M_ReadResults : BOOL

VAR
	DelayReadata: TON;
END_VAR
M_ReadResults:=FALSE;

Readcase:=0;
bReadBusy:=in_bOut3Results;


CASE Readcase OF
	
		0:
			IF in_bReadComplete THEN
				
			MEMSET(destAddr:=ADR(out_strReadData) , fillByte:=0 , n:=SIZEOF(out_strReadData) );
			DelayReadata(IN:=TRUE , PT:=T#200MS , Q=> , ET=> );
			IF DelayReadata.Q THEN
			Readcase:=1;
			Test:=TRUE;		
			END_IF

			END_IF			

		1:
			MEMCPY(destAddr:=ADR(out_strReadData) , srcAddr:=ADR(in_arrReadData) , n:=in_uintReadDataSize );

			DelayReadata(IN:=FALSE , PT:= , Q=> , ET=> );

			IF in_bOut1Results THEN
			Out_BarcodeReadGood:=TRUE;
			END_IF

			IF in_bOut2Results THEN
			out_BarcodeReadBadORError:=TRUE;
			END_IF
						

			
	
END_CASE
END_METHOD

(* This should clear any errors on the device and bring it to a state where
	it is ready to be energized or otherwise activated. *)
METHOD M_Reset : BOOL
M_Reset:=FALSE;
ResetCase:=0;	

CASE ResetCase OF
		0:
			IF bReset THEN
				bResetBusy:=TRUE;
				TriggerCounter.RESET:=FALSE;
				PresetTrig(CLK:=FALSE , Q=> );
				Out_BarcodeReadGood:=FALSE;
				out_BarcodeReadBadORError:=FALSE;
//				Out_BarcodeReadError:=FALSE;	
				b_BusyTrigger:=false;				
				ResetCase:=1;
			END_IF			

		1:
			out_ErrorClear:=TRUE;
			out_ReadCompleteClear:=TRUE;
			out_PresetCompleteClear:=TRUE;
			out_EXTRequestCompleteClear:=TRUE;
			Out_RegisterPresetClearDataAvailable:=TRUE;
			PresetTimerReq(IN:=TRUE ,PT:=T#500MS , Q=> , ET=> );	
			b_BusyTrigger:=TRUE;
			IF PresetTimerReq.Q THEN
			ResetCase:=2;
			END_IF

		2:	
			out_ErrorClear:=FALSE;
			out_ReadCompleteClear:=FALSE;
			out_PresetCompleteClear:=FALSE;
			out_EXTRequestCompleteClear:=FALSE;
			Out_RegisterPresetClearDataAvailable:=FALSE;
			bResetBusy:=FALSE;
			PresetTimerReq(IN:=FALSE ,PT:= , Q=> , ET=> );	
			ResetCase:=0;	
END_CASE
END_METHOD

(* This should move the program state from whatever state it is in to the
	Running state, and then return TRUE once successful. Starting from the
	Paused state should always continue execution from whatever point the
	program was at when the program was initially paused. *)
METHOD M_StartProgram : BOOL
END_METHOD

(* This should change the program state from whatever state it was in to the
	Stopped state and then return TRUE. Moving to the Stopped state should
	always reset the program execution back to the beginning. *)
METHOD M_StopProgram : BOOL
END_METHOD

METHOD M_Trigger : BOOL


VAR
END_VAR
M_Trigger:=FALSE;
TriggerCAse:=0;

out_bReadRequest :=bTrigger;

CASE TriggerCase OF
	0:IF bTrigger THEN
		out_bReadRequest:=TRUE;
		b_BusyTrigger:=TRUE;
		CaeraTrigDelay(IN:=TRUE , PT:=T#200MS , Q=> , ET=> );
		END_IF
		IF CaeraTrigDelay.Q THEN
			TriggerCase:=1;
		END_IF	
	1:	
		out_bReadRequest:=FALSE;
		CaeraTrigDelay(IN:=FALSE , PT:= , Q=> , ET=> );
		TriggerCase:=0;
		b_BusyTrigger:=FALSE;
END_CASE
END_METHOD

(* This property should be TRUE while any method in this interface is actively
	executing, or FALSE otherwise. *)
PROPERTY P_bEnableBusy : BOOL
GET
END_GET
END_PROPERTY

(* This should be set to TRUE if M_Enable is successful or M_GetEnableStatus
	determines the device to be enabled, and set to FALSE if M_Disable is
	called at all, M_GetEnableStatus fails, or M_GetEnableStatus determines
	the device to be not enabled. *)
PROPERTY P_bEnabled : BOOL
GET
END_GET
END_PROPERTY

(* This property should be TRUE while any method in this interface is actively
	executing, or FALSE otherwise. *)
PROPERTY P_bProgramControlBusy : BOOL
GET
END_GET
END_PROPERTY

PROPERTY P_bReadBusy : BOOL
GET
P_bReadBusy:=bReadBusy;
END_GET
END_PROPERTY


(* This property should be TRUE while any method in this interface is actively
	executing, or FALSE otherwise. *)
PROPERTY P_bResetBusy : BOOL
GET
P_bResetBusy:=bResetBusy;
END_GET
END_PROPERTY

PROPERTY P_bResultsAvailable : BOOL
GET
P_bResultsAvailable:=in_bResultDataAvailable;
END_GET
END_PROPERTY


PROPERTY P_bTriggerBusy : BOOL
GET
P_bTriggerBusy:=b_BusyTrigger;
END_GET
END_PROPERTY

(* The current E_ProgramState value of the device. This should be reset to
	E_ProgramState.Unknown if any methods in this interface interact with the
	device but fail. *)
PROPERTY P_enumProgramState : Sensata_Common.E_ProgramState
GET
END_GET
END_PROPERTY

(* The value of the currently loaded program. This should only be set by
	M_LoadProgram or M_GetCurrentProgram, and set to a blank string if either
	fail. *)
PROPERTY P_strCurrentProgram : Sensata_Common.T_MaxString
GET
END_GET
END_PROPERTY

PROPERTY P_strDescription : Sensata_Common.T_MaxString
GET
P_strDescription := 'Keyence SR751';
END_GET
END_PROPERTY

PROPERTY P_strMake : Sensata_Common.T_MaxString
GET
P_strMake := 'Keyence';
END_GET
END_PROPERTY

PROPERTY P_strModel : Sensata_Common.T_MaxString
GET
P_strModel := 'SR751';
END_GET
END_PROPERTY

PROPERTY P_strVersion : Sensata_Common.T_MaxString
GET
END_GET
END_PROPERTY

END_FUNCTION_BLOCK

// Concrete/Keyence/SR Series/FB_KeyenceSR
FUNCTION_BLOCK FB_KeyenceSR EXTENDS FB_BarcodeReader
	IMPLEMENTS I_Triggerable, I_Readable, I_Resettable
VAR_INPUT
	in_bHandshakeEnabled: BOOL;
	
	in_bTriggerBusy: BOOL;
	
	in_bReadComplete: BOOL;
	in_uintReadDataSize: UINT;
	in_arrReadData: ARRAY[0..127] OF BYTE;
	in_bReadDataAvailable: BOOL;
	in_bReadDataComplete: BOOL;
	in_intReadDataUpdateCount: INT;
	in_intReadDataReadyCount: INT;
	in_bReadError: BOOL;
END_VAR
VAR_OUTPUT
	out_bClear: BOOL;
	out_bReadRequest: BOOL;
	out_bReadCompleteClear: BOOL;
	out_bReadDataUpdate: BOOL;
	out_strReadData: STRING(127);
END_VAR
VAR
	bTriggeringBusy: BOOL;
	intTriggerStep: INT;
	bReadBusy: BOOL;
	intReadStep: INT;
	intClearStep: INT;
	
	bReadResultBusy: BOOL;
	bTriggerBusy: BOOL;
	bClearBusy: BOOL;
END_VAR

A_CommandRecovery();

(* Clears all results currently available on the camera. *)
METHOD M_ClearResults : BOOL
VAR_INST // added by the converter: edge detectors and wires of the graphical bodies
    _w1, _w2, _w3, _w4 : BOOL;
END_VAR
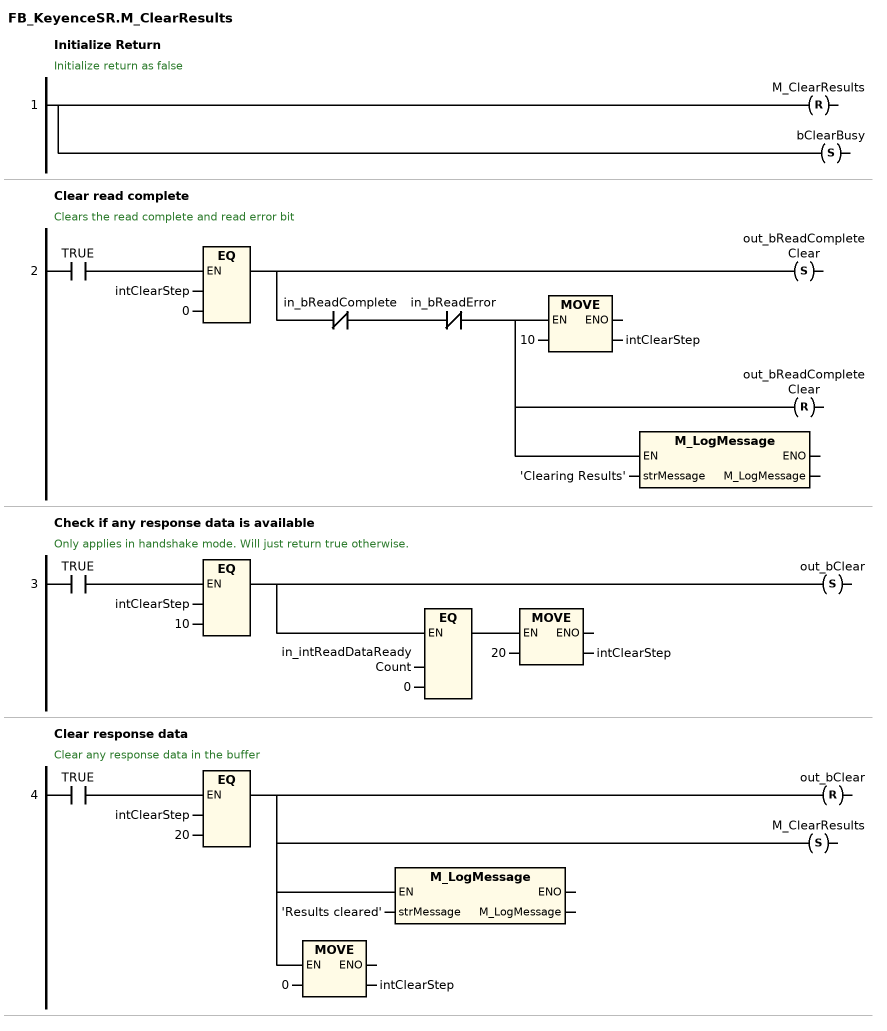
// NETWORK 1: Initialize Return
// Initialize return as false
M_ClearResults R= TRUE;
bClearBusy S= TRUE;

// NETWORK 2: Clear read complete
// Clears the read complete and read error bit
_w1 := intClearStep = 0;
out_bReadCompleteClear S= _w1;
_w2 := _w1 AND NOT in_bReadComplete AND NOT in_bReadError;
IF _w2 THEN intClearStep := 10; END_IF
out_bReadCompleteClear R= _w2;
IF _w2 THEN M_LogMessage(strMessage := 'Clearing Results'); END_IF

// NETWORK 3: Check if any response data is available
// Only applies in handshake mode. Will just return true otherwise.
_w3 := intClearStep = 10;
out_bClear S= _w3;
IF _w3 AND in_intReadDataReadyCount = 0 THEN intClearStep := 20; END_IF

// NETWORK 4: Clear response data
// Clear any response data in the buffer
_w4 := intClearStep = 20;
out_bClear R= _w4;
M_ClearResults S= _w4;
IF _w4 THEN M_LogMessage(strMessage := 'Results cleared'); END_IF
IF _w4 THEN intClearStep := 0; END_IF
END_METHOD

(* Reads one result from the camera. *)
METHOD M_ReadResult : BOOL
VAR_INST // added by the converter: edge detectors and wires of the graphical bodies
    _w1, _w2, _w3, _w4, _w5, _w6, _w7, _w8, _w9, _w10 : BOOL;
END_VAR
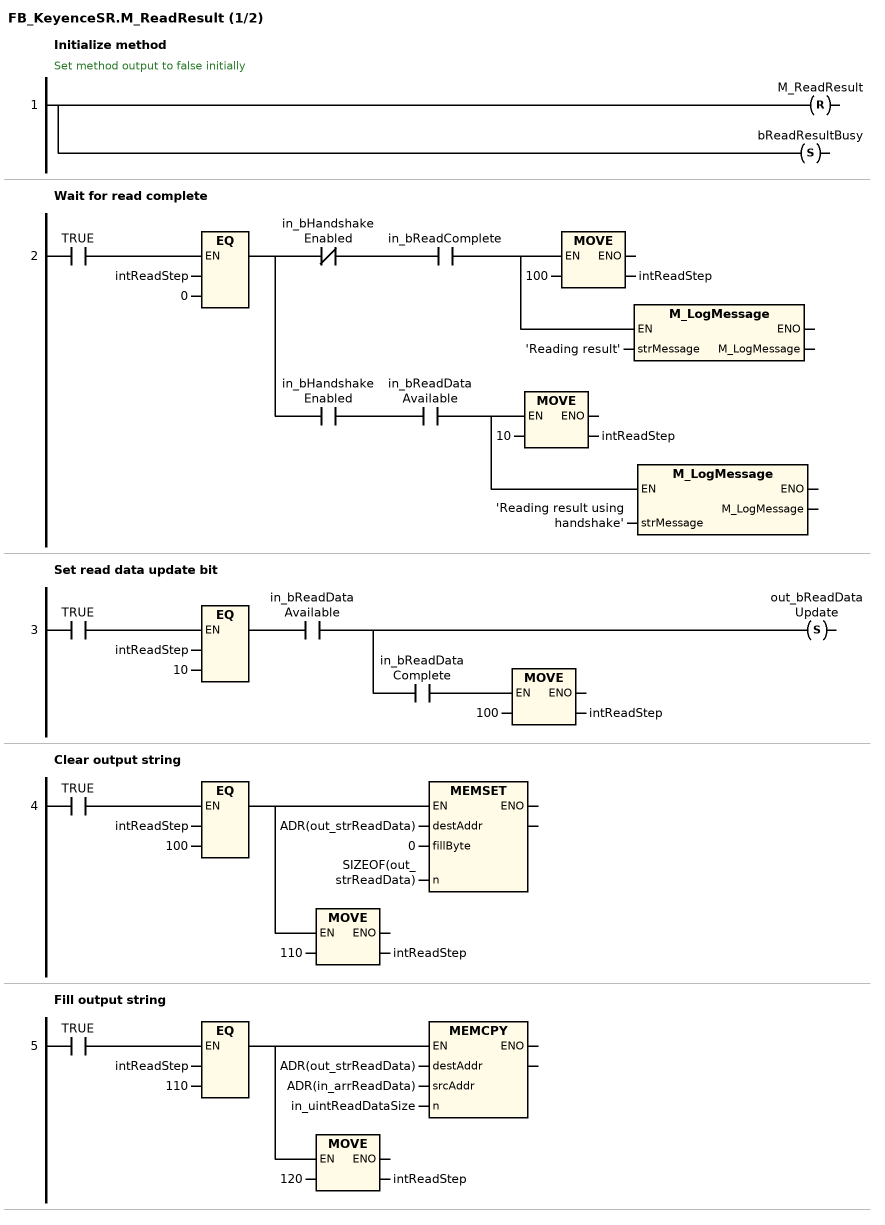
// NETWORK 1: Initialize method
// Set method output to false initially
M_ReadResult R= TRUE;
bReadResultBusy S= TRUE;

// NETWORK 2: Wait for read complete
_w1 := intReadStep = 0;
_w2 := _w1 AND NOT in_bHandshakeEnabled AND in_bReadComplete;
IF _w2 THEN intReadStep := 100; END_IF
IF _w2 THEN M_LogMessage(strMessage := 'Reading result'); END_IF
_w3 := _w1 AND in_bHandshakeEnabled AND in_bReadDataAvailable;
IF _w3 THEN intReadStep := 10; END_IF
IF _w3 THEN M_LogMessage(strMessage := 'Reading result using handshake'); END_IF

// NETWORK 3: Set read data update bit
_w4 := intReadStep = 10 AND in_bReadDataAvailable;
out_bReadDataUpdate S= _w4;
IF _w4 AND in_bReadDataComplete THEN intReadStep := 100; END_IF

// NETWORK 4: Clear output string
_w5 := intReadStep = 100;
IF _w5 THEN MEMSET(destAddr := ADR(out_strReadData), fillByte := 0, n := SIZEOF(out_strReadData)); END_IF
IF _w5 THEN intReadStep := 110; END_IF

// NETWORK 5: Fill output string
_w6 := intReadStep = 110;
IF _w6 THEN
    MEMCPY(destAddr := ADR(out_strReadData), srcAddr := ADR(in_arrReadData), n := in_uintReadDataSize);
END_IF
IF _w6 THEN intReadStep := 120; END_IF

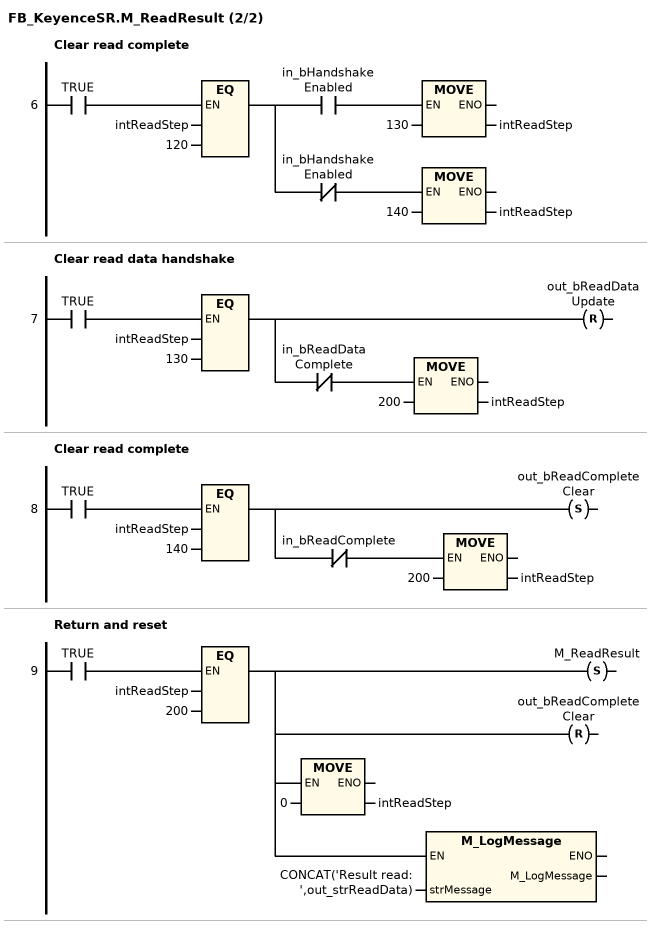
// NETWORK 6: Clear read complete
_w7 := intReadStep = 120;
IF _w7 AND in_bHandshakeEnabled THEN intReadStep := 130; END_IF
IF _w7 AND NOT in_bHandshakeEnabled THEN intReadStep := 140; END_IF

// NETWORK 7: Clear read data handshake
_w8 := intReadStep = 130;
out_bReadDataUpdate R= _w8;
IF _w8 AND NOT in_bReadDataComplete THEN intReadStep := 200; END_IF

// NETWORK 8: Clear read complete
_w9 := intReadStep = 140;
out_bReadCompleteClear S= _w9;
IF _w9 AND NOT in_bReadComplete THEN intReadStep := 200; END_IF

// NETWORK 9: Return and reset
_w10 := intReadStep = 200;
M_ReadResult S= _w10;
out_bReadCompleteClear R= _w10;
IF _w10 THEN intReadStep := 0; END_IF
IF _w10 THEN M_LogMessage(strMessage := CONCAT('Result read: ',out_strReadData)); END_IF
END_METHOD

(* True while this interface is busy. *)
PROPERTY P_bReadBusy : BOOL
GET
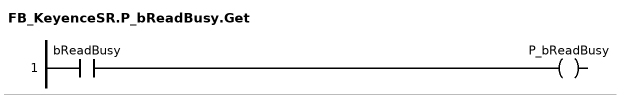
// NETWORK 1
P_bReadBusy := bReadBusy;
END_GET
END_PROPERTY

(* True if there are results available. *)
PROPERTY P_bResultsAvailable : BOOL
GET
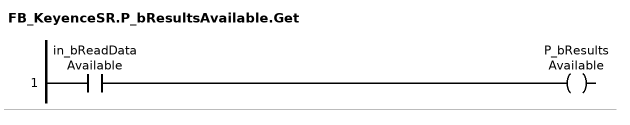
// NETWORK 1
P_bResultsAvailable := in_bReadDataAvailable;
END_GET
END_PROPERTY

(* This should clear any errors on the device and bring it to a state where
	it is ready to be energized or otherwise activated. *)
METHOD M_Reset : BOOL
VAR_INST // added by the converter: edge detectors and wires of the graphical bodies
    _w1 : BOOL;
END_VAR
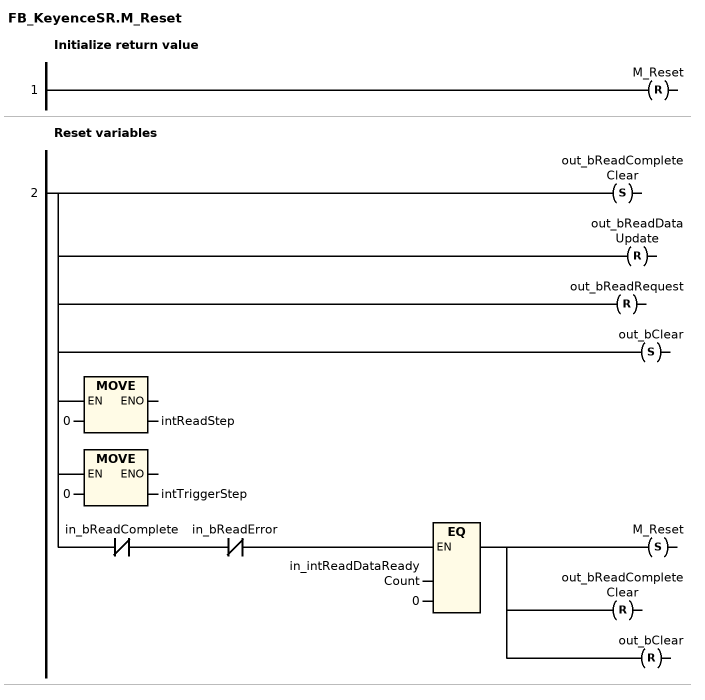
// NETWORK 1: Initialize return value
M_Reset R= TRUE;

// NETWORK 2: Reset variables
out_bReadCompleteClear S= TRUE;
out_bReadDataUpdate R= TRUE;
out_bReadRequest R= TRUE;
out_bClear S= TRUE;
intReadStep := 0;
intTriggerStep := 0;
_w1 := NOT in_bReadComplete AND NOT in_bReadError AND in_intReadDataReadyCount = 0;
M_Reset S= _w1;
out_bReadCompleteClear R= _w1;
out_bClear R= _w1;
END_METHOD

(* This property should be TRUE while any method in this interface is actively
	executing, or FALSE otherwise. *)
PROPERTY P_bResetBusy : BOOL
GET
// NETWORK 1
END_GET
END_PROPERTY

(*
Triggers the function block.
*)
METHOD M_Trigger : BOOL
VAR
	_bErrorSet: BOOL;
END_VAR
VAR_INST // added by the converter: edge detectors and wires of the graphical bodies
    _w1, _w2, _w3, _w4, _w5 : BOOL;
END_VAR
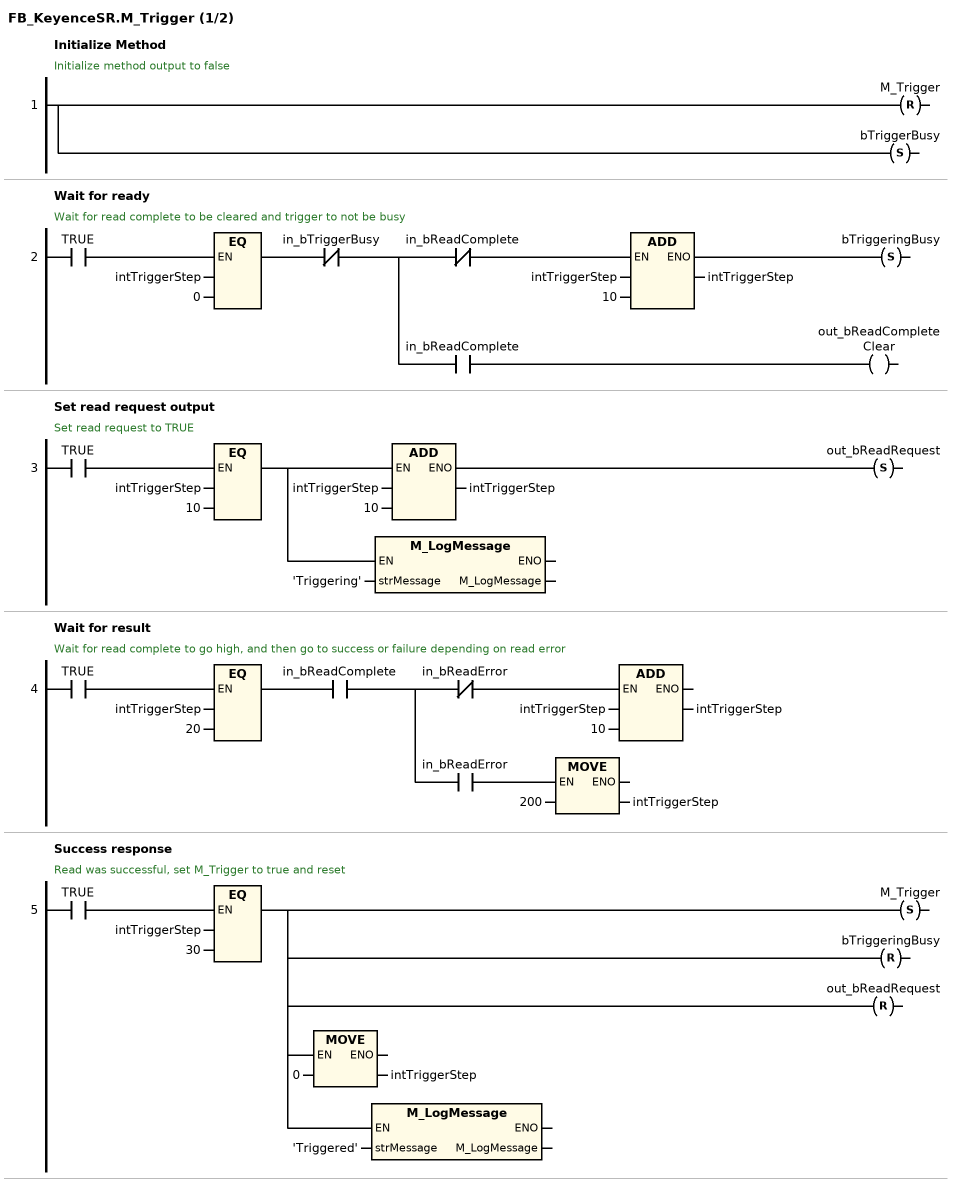
// NETWORK 1: Initialize Method
// Initialize method output to false
M_Trigger R= TRUE;
bTriggerBusy S= TRUE;

// NETWORK 2: Wait for ready
// Wait for read complete to be cleared and trigger to not be busy
_w1 := intTriggerStep = 0 AND NOT in_bTriggerBusy;
IF _w1 AND NOT in_bReadComplete THEN intTriggerStep := intTriggerStep + 10; END_IF
bTriggeringBusy S= _w1 AND NOT in_bReadComplete;
out_bReadCompleteClear := _w1 AND in_bReadComplete;

// NETWORK 3: Set read request output
// Set read request to TRUE
_w2 := intTriggerStep = 10;
IF _w2 THEN intTriggerStep := intTriggerStep + 10; END_IF
out_bReadRequest S= _w2;
IF _w2 THEN M_LogMessage(strMessage := 'Triggering'); END_IF

// NETWORK 4: Wait for result
// Wait for read complete to go high, and then go to success or failure depending on read error
_w3 := intTriggerStep = 20 AND in_bReadComplete;
IF _w3 AND NOT in_bReadError THEN intTriggerStep := intTriggerStep + 10; END_IF
IF _w3 AND in_bReadError THEN intTriggerStep := 200; END_IF

// NETWORK 5: Success response
// Read was successful, set M_Trigger to true and reset
_w4 := intTriggerStep = 30;
M_Trigger S= _w4;
bTriggeringBusy R= _w4;
out_bReadRequest R= _w4;
IF _w4 THEN intTriggerStep := 0; END_IF
IF _w4 THEN M_LogMessage(strMessage := 'Triggered'); END_IF

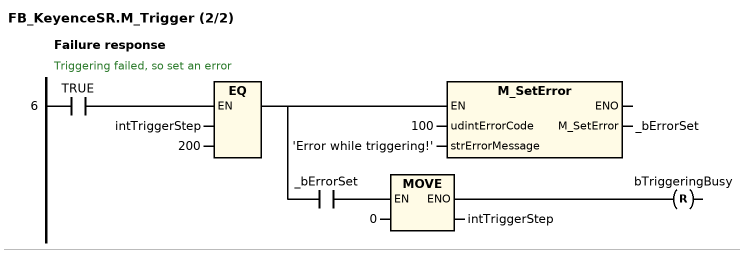
// NETWORK 6: Failure response
// Triggering failed, so set an error
_w5 := intTriggerStep = 200;
IF _w5 THEN _bErrorSet := M_SetError(udintErrorCode := 100, strErrorMessage := 'Error while triggering!'); END_IF
IF _w5 AND _bErrorSet THEN intTriggerStep := 0; END_IF
bTriggeringBusy R= _w5 AND _bErrorSet;
END_METHOD

(*
Stays high while the function block is performing the tasks that were triggered.
*)
PROPERTY P_bTriggerBusy : BOOL
GET
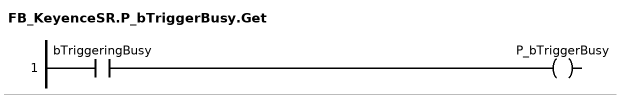
// NETWORK 1
P_bTriggerBusy := bTriggeringBusy;
END_GET
END_PROPERTY

ACTION A_ClearOutputs:
out_bClear:=FALSE;
out_bReadRequest:=FALSE;
out_bReadCompleteClear:=FALSE;
out_bReadDataUpdate:=FALSE;
END_ACTION

ACTION A_CommandRecovery:
IF NOT bReadResultBusy AND intReadStep > 0 THEN
	intReadStep := 0;
	A_ClearOutputs();
	THIS^.M_LogWarning('M_ReadResult ended prematurely!');
END_IF
bReadResultBusy := FALSE;

IF NOT bTriggerBusy AND intTriggerStep > 0 THEN
	intTriggerStep := 0;
	A_ClearOutputs();
	THIS^.M_LogWarning('M_Trigger ended prematurely!');
END_IF
bTriggerBusy := FALSE;

IF NOT bClearBusy AND intClearStep > 0 THEN
	intClearStep := 0;
	A_ClearOutputs();
	THIS^.M_LogWarning('M_Clear ended prematurely!');
END_IF
bClearBusy := FALSE;
END_ACTION

END_FUNCTION_BLOCK

// Concrete/Keyence/SR Series/FB_KeyenceNL20_EIP
FUNCTION_BLOCK FB_KeyenceNL20_EIP EXTENDS FB_BarcodeReader
	IMPLEMENTS I_Triggerable, I_Readable, I_Resettable
VAR_INPUT
	(* Set to TRUE if handshake is enabled in AutoID. *)
	in_bHandshakeEnabled: BOOL;
END_VAR
VAR_IN_OUT
	stIO: ST_KeyenceNL20_EIP;
END_VAR
VAR_OUTPUT
	out_strReadData: STRING(127);
END_VAR
VAR
	fbSR: FB_KeyenceSR;
	
	// INPUTS
	bTriggerBusy: BOOL;
	bReadComplete: BOOL;
	bReadError: BOOL;
	bReadDataAvailable: BOOL;
	uintReadDataSize: UINT;
	arrReadData: ARRAY [0..127] OF BYTE;
	bReadDataComplete: BOOL;
	
	// OUTPUTS
	bReadRequest: BOOL;
	bReadCompleteClear: BOOL;
	bReadDataUpdate: BOOL;
	intReadDataUpdateCount: INT;
	intReadDataReadyCount: INT;
	bClear: BOOL;
END_VAR

// Map inputs
bTriggerBusy := FALSE;
bReadComplete := BIT_TO_BOOL(stIO.stIn.bitReadComplete);
bReadError := BIT_TO_BOOL(stIO.stIn.bitOUT2Status);
bReadDataAvailable := BIT_TO_BOOL(stIO.stIn.bitResponseDataAvailable);
bReadDataComplete := BIT_TO_BOOL(stIO.stIn.bitResultDataStrobe);
uintReadDataSize := stIO.stIn.uintResultDataSize;
arrReadData := stIO.stIn.arrResultData;
intReadDataReadyCount := UINT_TO_INT(stIO.stIn.uintResultDataReadyCount);
intReadDataUpdateCount:= UINT_TO_INT(stIO.stIn.uintResultDataUpdateCount);

// Call FB
A_SR();

// Map outputs
stIO.stOut.bitReadRequest := BOOL_TO_BIT(bReadRequest);
stIO.stOut.bitReadCompleteClear := BOOL_TO_BIT(bReadCompleteClear);
stIO.stOut.bitResultDataLatch := BOOL_TO_BIT(bReadDataUpdate);
stIO.stOut.bitErrorClear := BOOL_TO_BIT(bClear);

ACTION A_SR:
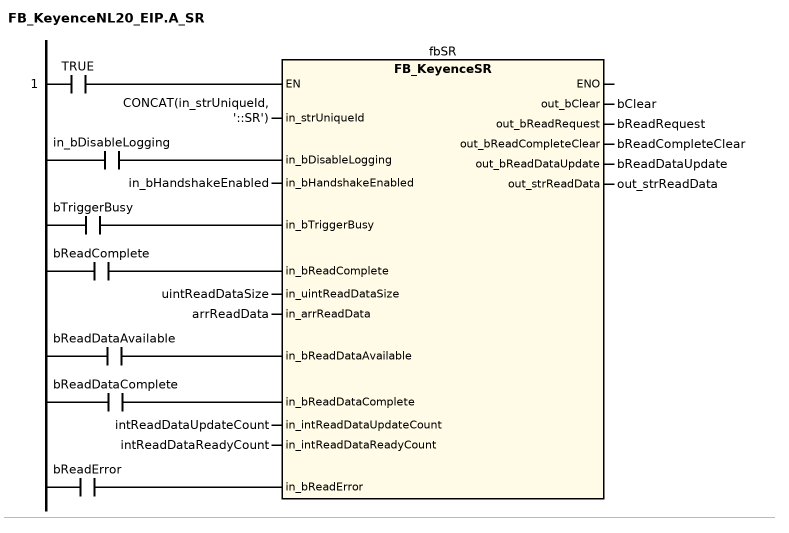
// NETWORK 1
fbSR(
    in_strUniqueId := CONCAT(in_strUniqueId,'::SR'),
    in_bDisableLogging := in_bDisableLogging,
    in_bHandshakeEnabled := in_bHandshakeEnabled,
    in_bTriggerBusy := bTriggerBusy,
    in_bReadComplete := bReadComplete,
    in_uintReadDataSize := uintReadDataSize,
    in_arrReadData := arrReadData,
    in_bReadDataAvailable := bReadDataAvailable,
    in_bReadDataComplete := bReadDataComplete,
    in_intReadDataUpdateCount := intReadDataUpdateCount,
    in_intReadDataReadyCount := intReadDataReadyCount,
    in_bReadError := bReadError,
    out_bClear => bClear,
    out_bReadRequest => bReadRequest,
    out_bReadCompleteClear => bReadCompleteClear,
    out_bReadDataUpdate => bReadDataUpdate,
    out_strReadData => out_strReadData); // FB_KeyenceSR
END_ACTION

(* Clears all results currently available on the camera. *)
METHOD M_ClearResults : BOOL
M_ClearResults := fbSR.M_ClearResults();
IF fbSR.P_bError THEN
	THIS^.M_SetError(fbSR.P_udintErrorCode, 'Error on SR block!');
END_IF
END_METHOD

(* Reads one result from the camera. *)
METHOD M_ReadResult : BOOL
M_ReadResult := fbSR.M_ReadResult();
IF fbSR.P_bError THEN
	THIS^.M_SetError(fbSR.P_udintErrorCode, 'Error on SR block!');
END_IF
END_METHOD

(* This should clear any errors on the device and bring it to a state where
	it is ready to be energized or otherwise activated. *)
METHOD M_Reset : BOOL
fbSR.M_ClearError();
M_Reset := fbSR.M_Reset();
IF fbSR.P_bError THEN
	THIS^.M_SetError(fbSR.P_udintErrorCode, 'Error on SR block!');
END_IF
END_METHOD

(*
Triggers the function block.
*)
METHOD M_Trigger : BOOL
M_Trigger := fbSR.M_Trigger();
IF fbSR.P_bError THEN
	THIS^.M_SetError(fbSR.P_udintErrorCode, 'Error on SR block!');
END_IF
END_METHOD

(* True while this interface is busy. *)
PROPERTY P_bReadBusy : BOOL
GET
P_bReadBusy := fbSR.P_bReadBusy;
END_GET
END_PROPERTY

(* This property should be TRUE while any method in this interface is actively
	executing, or FALSE otherwise. *)
PROPERTY P_bResetBusy : BOOL
GET
P_bResetBusy := fbSR.P_bResetBusy;
END_GET
END_PROPERTY

(* True if there are results available. *)
PROPERTY P_bResultsAvailable : BOOL
GET
P_bResultsAvailable := fbSR.P_bResultsAvailable;
END_GET
END_PROPERTY

(*
Stays high while the function block is performing the tasks that were triggered.
*)
PROPERTY P_bTriggerBusy : BOOL
GET
P_bTriggerBusy := fbSR.P_bTriggerBusy;
END_GET
END_PROPERTY

END_FUNCTION_BLOCK

// Concrete/Keyence/SR Series/FB_KeyenceSR750_EIP
FUNCTION_BLOCK FB_KeyenceSR750_EIP EXTENDS FB_BarcodeReader
	IMPLEMENTS I_Triggerable, I_Readable, I_Resettable
VAR_INPUT
	(* Set to TRUE if handshake is enabled in AutoID. *)
	in_bHandshakeEnabled: BOOL;
	(* If one of the programmable outputs is set to ERROR or NG,
		set this to the number of that output (Typically 2) *)
	in_uintErrorInput: UINT := 0;
END_VAR
VAR_IN_OUT
	stIO: ST_KeyenceSR750_EIP;
END_VAR
VAR_OUTPUT
	out_strReadData: STRING(127);
END_VAR
VAR
	fbSR: FB_KeyenceSR;
	
	// INPUTS
	bTriggerBusy: BOOL;
	bReadComplete: BOOL;
	bReadError: BOOL;
	bReadDataAvailable: BOOL;
	uintReadDataSize: UINT;
	arrReadData: ARRAY [0..127] OF BYTE;
	bReadDataComplete: BOOL;
	
	// OUTPUTS
	bReadRequest: BOOL;
	bReadCompleteClear: BOOL;
	bReadDataUpdate: BOOL;
	intReadDataReadyCount: INT;
	intReadDataUpdateCount: INT;
	bClear: BOOL;
END_VAR

// Map inputs
bTriggerBusy := BIT_TO_BOOL(stIO.stIn.bitTrgBusy);
bReadComplete := BIT_TO_BOOL(stIO.stIn.bitReadComplete);
CASE in_uintErrorInput OF
	1: bReadError := BIT_TO_BOOL(stIO.stIn.bitReadFailure) OR BIT_TO_BOOL(stIO.stIn.bitOUT1Status);
	2: bReadError := BIT_TO_BOOL(stIO.stIn.bitReadFailure) OR BIT_TO_BOOL(stIO.stIn.bitOUT2Status);
	3: bReadError := BIT_TO_BOOL(stIO.stIn.bitReadFailure) OR BIT_TO_BOOL(stIO.stIn.bitOUT3Status);
ELSE
	bReadError := BIT_TO_BOOL(stIO.stIn.bitReadFailure);
END_CASE
bReadDataAvailable := BIT_TO_BOOL(stIO.stIn.bitResponseDataAvailable);
bReadDataComplete := BIT_TO_BOOL(stIO.stIn.bitResultDataStrobe);
uintReadDataSize := stIO.stIn.uintResultDataSize;
arrReadData := stIO.stIn.arrResultData;
intReadDataReadyCount := UINT_TO_INT(stIO.stIn.uintResultDataReadyCount);
intReadDataUpdateCount:= UINT_TO_INT(stIO.stIn.uintResultDataUpdateCount);


// Map outputs
stIO.stOut.bitReadRequest := BOOL_TO_BIT(bReadRequest);
stIO.stOut.bitReadCompleteClear := BOOL_TO_BIT(bReadCompleteClear);
stIO.stOut.bitResultDataLatch := BOOL_TO_BIT(bReadDataUpdate);
stIO.stOut.bitErrorClear := BOOL_TO_BIT(bClear);

// Call FB
A_SR();

ACTION A_SR:
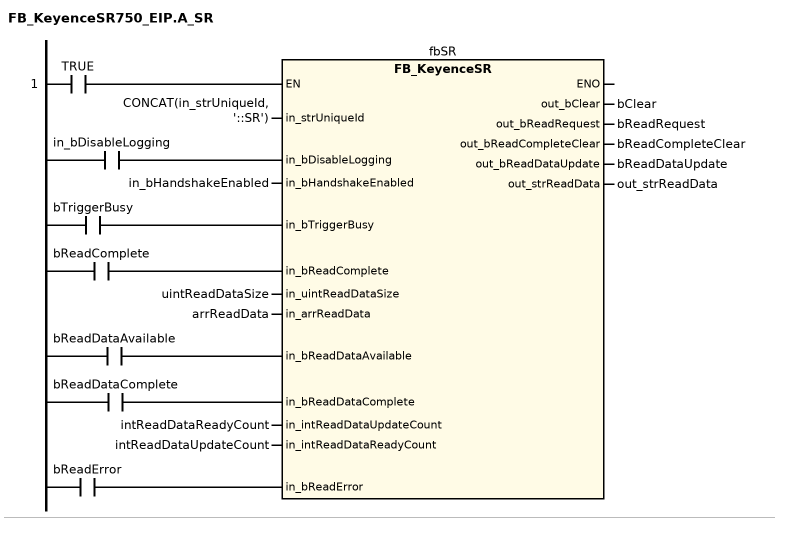
// NETWORK 1
fbSR(
    in_strUniqueId := CONCAT(in_strUniqueId,'::SR'),
    in_bDisableLogging := in_bDisableLogging,
    in_bHandshakeEnabled := in_bHandshakeEnabled,
    in_bTriggerBusy := bTriggerBusy,
    in_bReadComplete := bReadComplete,
    in_uintReadDataSize := uintReadDataSize,
    in_arrReadData := arrReadData,
    in_bReadDataAvailable := bReadDataAvailable,
    in_bReadDataComplete := bReadDataComplete,
    in_intReadDataUpdateCount := intReadDataReadyCount,
    in_intReadDataReadyCount := intReadDataUpdateCount,
    in_bReadError := bReadError,
    out_bClear => bClear,
    out_bReadRequest => bReadRequest,
    out_bReadCompleteClear => bReadCompleteClear,
    out_bReadDataUpdate => bReadDataUpdate,
    out_strReadData => out_strReadData); // FB_KeyenceSR
END_ACTION

(* Clears all results currently available on the camera. *)
METHOD M_ClearResults : BOOL
M_ClearResults := fbSR.M_ClearResults();
IF fbSR.P_bError THEN
	THIS^.M_SetError(fbSR.P_udintErrorCode, 'Error on SR block!');
END_IF
END_METHOD

(* Reads one result from the camera. *)
METHOD M_ReadResult : BOOL
M_ReadResult := fbSR.M_ReadResult();
IF fbSR.P_bError THEN
	THIS^.M_SetError(fbSR.P_udintErrorCode, 'Error on SR block!');
END_IF
END_METHOD

(* This should clear any errors on the device and bring it to a state where
	it is ready to be energized or otherwise activated. *)
METHOD M_Reset : BOOL
fbSR.M_ClearError();
M_Reset := fbSR.M_Reset();
IF fbSR.P_bError THEN
	THIS^.M_SetError(fbSR.P_udintErrorCode, 'Error on SR block!');
END_IF
END_METHOD

(*
Triggers the function block.
*)
METHOD M_Trigger : BOOL
M_Trigger := fbSR.M_Trigger();
IF fbSR.P_bError THEN
	THIS^.M_SetError(fbSR.P_udintErrorCode, 'Error on SR block!');
END_IF
END_METHOD

(* True while this interface is busy. *)
PROPERTY P_bReadBusy : BOOL
GET
P_bReadBusy := fbSR.P_bReadBusy;
END_GET
END_PROPERTY

(* This property should be TRUE while any method in this interface is actively
	executing, or FALSE otherwise. *)
PROPERTY P_bResetBusy : BOOL
GET
P_bResetBusy := fbSR.P_bResetBusy;
END_GET
END_PROPERTY

(* True if there are results available. *)
PROPERTY P_bResultsAvailable : BOOL
GET
P_bResultsAvailable := fbSR.P_bResultsAvailable;
END_GET
END_PROPERTY

(*
Stays high while the function block is performing the tasks that were triggered.
*)
PROPERTY P_bTriggerBusy : BOOL
GET
P_bTriggerBusy := fbSR.P_bTriggerBusy;
END_GET
END_PROPERTY

END_FUNCTION_BLOCK

// Concrete/Keyence/SR Series/FB_KeyenceSRX1H3H_EIP
FUNCTION_BLOCK FB_KeyenceSRX1H3H_EIP EXTENDS FB_BarcodeReader
	IMPLEMENTS I_Triggerable, I_Readable, I_Resettable
VAR_INPUT
	(* Set to TRUE if handshake is enabled in AutoID. *)
	in_bHandshakeEnabled: BOOL;
	(* If one of the programmable outputs is set to ERROR or NG,
		set this to the number of that output (Typically 2) *)
	in_uintErrorInput: UINT := 0;
END_VAR
VAR_IN_OUT
	stIO: ST_KeyenceSRX1H3H_EIP;
END_VAR
VAR_OUTPUT
	(* Barcode that was read. *)
	out_strReadData: STRING(127);
END_VAR
VAR
	fbSR: FB_KeyenceSR;
	
	// INPUTS
	bTriggerBusy: BOOL;
	bReadComplete: BOOL;
	bReadError: BOOL;
	bReadDataAvailable: BOOL;
	uintReadDataSize: UINT;
	arrReadData: ARRAY [0..127] OF BYTE;
	bReadDataComplete: BOOL;
	
	// OUTPUTS
	bReadRequest: BOOL;
	bReadCompleteClear: BOOL;
	bReadDataUpdate: BOOL;
	intReadDataReadyCount: INT;
	intReadDataUpdateCount: INT;
	bClear: BOOL;
END_VAR

// Map inputs
bTriggerBusy := BIT_TO_BOOL(stIO.stIn.bitTrgBusy);
bReadComplete := BIT_TO_BOOL(stIO.stIn.bitReadComplete);
CASE in_uintErrorInput OF
	1: bReadError := BIT_TO_BOOL(stIO.stIn.bitReadFailure) OR BIT_TO_BOOL(stIO.stIn.bitOUT1Status);
	2: bReadError := BIT_TO_BOOL(stIO.stIn.bitReadFailure) OR BIT_TO_BOOL(stIO.stIn.bitOUT2Status);
	3: bReadError := BIT_TO_BOOL(stIO.stIn.bitReadFailure) OR BIT_TO_BOOL(stIO.stIn.bitOUT3Status);
ELSE
	bReadError := BIT_TO_BOOL(stIO.stIn.bitReadFailure);
END_CASE
bReadDataAvailable := BIT_TO_BOOL(stIO.stIn.bitResponseDataAvailable);
bReadDataComplete := BIT_TO_BOOL(stIO.stIn.bitResultDataStrobe);
uintReadDataSize := stIO.stIn.uintResultDataSize;
arrReadData := stIO.stIn.arrResultData;
intReadDataReadyCount := UINT_TO_INT(stIO.stIn.uintResultDataReadyCount);
intReadDataUpdateCount:= UINT_TO_INT(stIO.stIn.uintResultDataUpdateCount);


// Map outputs
stIO.stOut.bitReadRequest := BOOL_TO_BIT(bReadRequest);
stIO.stOut.bitReadCompleteClear := BOOL_TO_BIT(bReadCompleteClear);
stIO.stOut.bitResultDataLatch := BOOL_TO_BIT(bReadDataUpdate);
stIO.stOut.bitErrorClear := BOOL_TO_BIT(bClear);

// Call FB
A_SR();

ACTION A_SR:
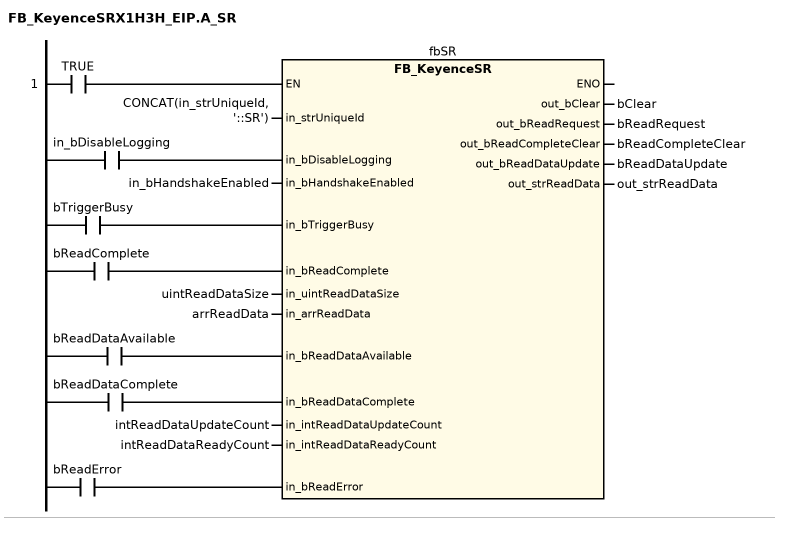
// NETWORK 1
fbSR(
    in_strUniqueId := CONCAT(in_strUniqueId,'::SR'),
    in_bDisableLogging := in_bDisableLogging,
    in_bHandshakeEnabled := in_bHandshakeEnabled,
    in_bTriggerBusy := bTriggerBusy,
    in_bReadComplete := bReadComplete,
    in_uintReadDataSize := uintReadDataSize,
    in_arrReadData := arrReadData,
    in_bReadDataAvailable := bReadDataAvailable,
    in_bReadDataComplete := bReadDataComplete,
    in_intReadDataUpdateCount := intReadDataUpdateCount,
    in_intReadDataReadyCount := intReadDataReadyCount,
    in_bReadError := bReadError,
    out_bClear => bClear,
    out_bReadRequest => bReadRequest,
    out_bReadCompleteClear => bReadCompleteClear,
    out_bReadDataUpdate => bReadDataUpdate,
    out_strReadData => out_strReadData); // FB_KeyenceSR
END_ACTION

(* Clears all results currently available on the camera. *)
METHOD M_ClearResults : BOOL
M_ClearResults := fbSR.M_ClearResults();
IF fbSR.P_bError THEN
	THIS^.M_SetError(fbSR.P_udintErrorCode, 'Error on SR block!');
END_IF
END_METHOD

(* Reads one result from the camera. *)
METHOD M_ReadResult : BOOL
M_ReadResult := fbSR.M_ReadResult();
IF fbSR.P_bError THEN
	THIS^.M_SetError(fbSR.P_udintErrorCode, 'Error on SR block!');
END_IF
END_METHOD

(* This should clear any errors on the device and bring it to a state where
	it is ready to be energized or otherwise activated. *)
METHOD M_Reset : BOOL
fbSR.M_ClearError();
M_Reset := fbSR.M_Reset();
IF fbSR.P_bError THEN
	THIS^.M_SetError(fbSR.P_udintErrorCode, 'Error on SR block!');
END_IF
END_METHOD

(*
Triggers the function block.
*)
METHOD M_Trigger : BOOL
M_Trigger := fbSR.M_Trigger();
IF fbSR.P_bError THEN
	THIS^.M_SetError(fbSR.P_udintErrorCode, 'Error on SR block!');
END_IF
END_METHOD

(* True while this interface is busy. *)
PROPERTY P_bReadBusy : BOOL
GET
P_bReadBusy := fbSR.P_bReadBusy;
END_GET
END_PROPERTY

(* This property should be TRUE while any method in this interface is actively
	executing, or FALSE otherwise. *)
PROPERTY P_bResetBusy : BOOL
GET
P_bResetBusy := fbSR.P_bResetBusy;
END_GET
END_PROPERTY

(* True if there are results available. *)
PROPERTY P_bResultsAvailable : BOOL
GET
P_bResultsAvailable := fbSR.P_bResultsAvailable;
END_GET
END_PROPERTY

(*
Stays high while the function block is performing the tasks that were triggered.
*)
PROPERTY P_bTriggerBusy : BOOL
GET
P_bTriggerBusy := fbSR.P_bTriggerBusy;
END_GET
END_PROPERTY

END_FUNCTION_BLOCK

// Project Information/F_GetCompany
// This function has been automatically generated from the project information.
{attribute 'signature_flag' := '1073741824'}
{attribute 'TcGenerated'}
{attribute 'no-analysis'}
FUNCTION F_GetCompany : WSTRING
VAR_INPUT
	
END_VAR

F_GetCompany := "Sensata Technologies";

END_FUNCTION

// Project Information/F_GetTitle
// This function has been automatically generated from the project information.
{attribute 'signature_flag' := '1073741824'}
{attribute 'TcGenerated'}
{attribute 'no-analysis'}
FUNCTION F_GetTitle : WSTRING
VAR_INPUT
	
END_VAR

F_GetTitle := "Sensata_Vision";

END_FUNCTION

// Project Information/F_GetVersion
// This function has been automatically generated from the project information.
{attribute 'signature_flag' := '1073741824'}
{attribute 'TcGenerated'}
{attribute 'no-analysis'}
FUNCTION F_GetVersion : ST_LibVersion
VAR_INPUT
	
END_VAR

F_GetVersion.iMajor := 0;
F_GetVersion.iMinor := 0;
F_GetVersion.iBuild := 2;
F_GetVersion.iRevision := 0;

END_FUNCTION
